SPLINE
SPL {X  -144.515, Y  +305.495, Z    +0.000, E1   +74.543, E3 +104969.530}
SPL {X  -143.690, Y  +303.925, Z    +0.000, E1   +73.372, E3 +104980.269}
SPL {X  -141.993, Y  +300.823, Z    +0.000, E1   +72.659, E3 +104987.693}
SPL {X  -138.166, Y  +294.358, Z    +0.000, E1   +72.281, E3 +104994.155}
SPL {X  -134.385, Y  +288.571, Z    +0.000, E1   +71.826, E3 +105000.418}
SPL {X  -129.872, Y  +282.297, Z    +0.000, E1   +71.229, E3 +105007.588}
SPL {X  -124.448, Y  +275.510, Z    +0.000, E1   +70.509, E3 +105014.961}
SPL {X  -117.513, Y  +267.801, Z    +0.000, E1   +72.197, E3 +105012.544}
SPL {X   -63.140, Y  +230.421, Z    +0.000, E1   +55.875, E3 +105181.983}
ENDSPLINE

SPLINE
SPL {X  -130.329, Y  +282.905, Z    +0.000, E1   +55.659, E3 +105340.318}
SPL {X  -150.766, Y  +319.018, Z    +0.000, E1   +45.408, E3 +105348.811}
SPL {X  -157.479, Y  +339.138, Z    +0.000, E1   +35.556, E3 +105350.247}
SPL {X  -160.994, Y  +356.185, Z    +0.000, E1   +24.373, E3 +105352.293}
SPL {X  -162.352, Y  +368.168, Z    +0.000, E1   +14.282, E3 +105352.345}
SPL {X  -162.808, Y  +378.562, Z    +0.000, E1    +4.298, E3 +105352.277}
SPL {X  -162.820, Y  +382.500, Z    +0.000, E1    +0.000, E3 +105351.850}
SPL {X  -162.820, Y  +384.915, Z    +0.000, E1    -4.894, E3 +105351.563}
SPL {X  -162.820, Y  +388.986, Z    +0.000, E1   -15.047, E3 +105351.661}
SPL {X  -162.820, Y  +394.732, Z    +0.000, E1   -28.992, E3 +105351.512}
SPL {X  -162.820, Y  +403.075, Z    +0.000, E1   -46.096, E3 +105351.742}
SPL {X  -162.820, Y  +414.705, Z    +0.000, E1   -61.052, E3 +105351.188}
SPL {X  -162.820, Y  +466.149, Z    +0.000, E1   -74.732, E3 +105361.185}
SPL {X  -160.722, Y  +699.554, Z    +0.000, E1   -75.485, E3 +105458.595}
SPL {X  -159.966, Y  +703.854, Z    +0.000, E1   -74.386, E3 +105473.498}
SPL {X  -156.868, Y  +717.123, Z    +0.000, E1   -74.182, E3 +105483.176}
SPL {X  -153.226, Y  +728.564, Z    +0.000, E1   -73.755, E3 +105494.184}
SPL {X  -149.090, Y  +738.941, Z    +0.000, E1   -73.348, E3 +105503.758}
SPL {X  -145.714, Y  +746.149, Z    +0.000, E1   -72.951, E3 +105511.345}
SPL {X  -140.946, Y  +755.015, Z    +0.000, E1   -72.452, E3 +105520.447}
SPL {X  -136.902, Y  +761.638, Z    +0.000, E1   -71.857, E3 +105528.314}
SPL {X  -133.350, Y  +766.925, Z    +0.000, E1   -71.498, E3 +105533.635}
SPL {X  -129.687, Y  +771.946, Z    +0.000, E1   -71.061, E3 +105539.001}
SPL {X  -126.374, Y  +776.164, Z    +0.000, E1   -70.494, E3 +105544.254}
SPL {X  -122.717, Y  +780.508, Z    +0.000, E1   -70.361, E3 +105547.292}
SPL {X  -114.093, Y  +789.660, Z    +0.000, E1   -71.634, E3 +105547.310}
SPL {X   -61.593, Y  +824.220, Z    +0.000, E1   -55.970, E3 +105713.146}
ENDSPLINE

SPLINE
SPL {X  -131.598, Y  +769.376, Z    +0.000, E1   -56.871, E3 +105879.418}
SPL {X  -152.760, Y  +729.846, Z    +0.000, E1   -44.713, E3 +105886.470}
SPL {X  -158.868, Y  +709.157, Z    +0.000, E1   -33.466, E3 +105887.671}
SPL {X  -161.987, Y  +689.949, Z    +0.000, E1   -18.777, E3 +105888.632}
SPL {X  -162.803, Y  +675.860, Z    +0.000, E1    -4.958, E3 +105888.614}
SPL {X  -162.820, Y  +671.500, Z    +0.000, E1    +0.000, E3 +105888.151}
SPL {X  -162.820, Y  +669.410, Z    +0.000, E1    +4.515, E3 +105887.913}
SPL {X  -162.820, Y  +664.781, Z    +0.000, E1   +16.411, E3 +105887.908}
SPL {X  -162.820, Y  +659.650, Z    +0.000, E1   +29.778, E3 +105887.918}
SPL {X  -162.820, Y  +651.175, Z    +0.000, E1   +47.162, E3 +105888.068}
SPL {X  -162.820, Y  +637.134, Z    +0.000, E1   +65.232, E3 +105886.610}
SPL {X  -162.820, Y  +616.721, Z    +0.000, E1   +72.273, E3 +105890.344}
SPL {X  -162.820, Y  +577.172, Z    +0.000, E1   +75.843, E3 +105900.324}
SPL {X  -159.895, Y  +349.775, Z    +0.000, E1   +76.042, E3 +105991.990}
ENDSPLINE

SPLINE
SPL {X  -160.357, Y  +352.285, Z    +0.000, E1   +74.783, E3 +106004.928}
ENDSPLINE

SPLINE
SPL {X  -145.737, Y  +307.897, Z    +0.000, E1   +77.368, E3 +105997.503}
SPL {X  -145.329, Y  +307.084, Z    +0.000, E1   +76.571, E3 +106006.340}
ENDSPLINE

SPLINE
SPL {X  -145.355, Y  +307.136, Z    +0.000, E1   +75.607, E3 +106015.864}
ENDSPLINE

SPLINE
SPL {X  -144.515, Y  +305.495, Z    +0.000, E1   +74.543, E3 +106026.673}
SPL {X  -143.702, Y  +303.949, Z    +0.000, E1   +73.349, E3 +106037.595}
ENDSPLINE

SPLINE
SPL {X  -148.050, Y  +312.738, Z    +0.000, E1   +70.533, E3 +106054.970}
ENDSPLINE

SPLINE
SPL {X  -143.809, Y  +304.150, Z    +0.000, E1   +70.034, E3 +106064.386}
SPL {X  -139.938, Y  +297.268, Z    +0.000, E1   +69.438, E3 +106072.977}
SPL {X  -136.192, Y  +291.270, Z    +0.000, E1   +68.926, E3 +106080.124}
SPL {X  -131.963, Y  +285.127, Z    +0.000, E1   +68.405, E3 +106087.114}
SPL {X  -127.466, Y  +279.195, Z    +0.000, E1   +67.714, E3 +106094.402}
SPL {X  -119.204, Y  +269.591, Z    +0.000, E1   +69.726, E3 +106092.393}
SPL {X   -73.382, Y  +235.154, Z    +0.000, E1   +54.977, E3 +106258.070}
ENDSPLINE

SPLINE
SPL {X  -133.875, Y  +287.830, Z    +0.000, E1   +51.751, E3 +106397.273}
SPL {X  -153.240, Y  +325.474, Z    +0.000, E1   +39.999, E3 +106408.476}
SPL {X  -159.032, Y  +345.583, Z    +0.000, E1   +29.156, E3 +106408.960}
SPL {X  -161.304, Y  +358.334, Z    +0.000, E1   +20.524, E3 +106408.917}
SPL {X  -162.437, Y  +369.334, Z    +0.000, E1   +11.998, E3 +106410.096}
SPL {X  -162.814, Y  +379.161, Z    +0.000, E1    +3.343, E3 +106410.115}
SPL {X  -162.820, Y  +382.500, Z    +0.000, E1    +0.000, E3 +106409.598}
SPL {X  -162.820, Y  +384.390, Z    +0.000, E1    -3.279, E3 +106409.315}
SPL {X  -162.820, Y  +388.496, Z    +0.000, E1   -11.991, E3 +106409.217}
SPL {X  -162.820, Y  +392.944, Z    +0.000, E1   -22.020, E3 +106409.242}
SPL {X  -162.820, Y  +397.954, Z    +0.000, E1   -32.843, E3 +106409.282}
SPL {X  -162.820, Y  +404.232, Z    +0.000, E1   -44.157, E3 +106409.290}
SPL {X  -162.820, Y  +415.904, Z    +0.000, E1   -58.030, E3 +106409.563}
SPL {X  -162.820, Y  +472.155, Z    +0.000, E1   -74.123, E3 +106419.666}
SPL {X  -162.820, Y  +661.743, Z    +0.000, E1   -73.395, E3 +106514.800}
ENDSPLINE

SPLINE
SPL {X  -162.820, Y  +658.105, Z    +0.000, E1   -71.889, E3 +106528.198}
ENDSPLINE

SPLINE
SPL {X  -162.784, Y  +676.927, Z    +0.000, E1   -71.815, E3 +106541.726}
SPL {X  -161.514, Y  +694.081, Z    +0.000, E1   -71.845, E3 +106553.116}
SPL {X  -159.782, Y  +704.807, Z    +0.000, E1   -71.464, E3 +106564.098}
SPL {X  -157.050, Y  +716.463, Z    +0.000, E1   -71.316, E3 +106573.398}
SPL {X  -154.424, Y  +725.109, Z    +0.000, E1   -70.982, E3 +106582.250}
SPL {X  -151.195, Y  +733.918, Z    +0.000, E1   -70.611, E3 +106591.372}
SPL {X  -147.776, Y  +741.856, Z    +0.000, E1   -70.224, E3 +106599.820}
SPL {X  -144.623, Y  +748.297, Z    +0.000, E1   -69.772, E3 +106607.445}
SPL {X  -141.153, Y  +754.655, Z    +0.000, E1   -69.344, E3 +106614.749}
SPL {X  -137.365, Y  +760.914, Z    +0.000, E1   -68.751, E3 +106622.687}
SPL {X  -133.334, Y  +766.947, Z    +0.000, E1   -68.226, E3 +106629.792}
SPL {X  -129.138, Y  +772.665, Z    +0.000, E1   -67.631, E3 +106636.599}
SPL {X  -125.533, Y  +777.190, Z    +0.000, E1   -67.475, E3 +106640.296}
SPL {X   -73.826, Y  +818.621, Z    +0.000, E1   -58.574, E3 +106735.789}
ENDSPLINE

SPLINE
SPL {X  -110.901, Y  +792.711, Z    +0.000, E1   -55.300, E3 +106920.647}
SPL {X  -144.508, Y  +748.519, Z    +0.000, E1   -46.961, E3 +106945.683}
SPL {X  -158.446, Y  +710.986, Z    +0.000, E1   -30.228, E3 +106949.049}
SPL {X  -162.035, Y  +689.470, Z    +0.000, E1   -15.657, E3 +106950.620}
SPL {X  -162.788, Y  +676.746, Z    +0.000, E1    -5.020, E3 +106950.527}
SPL {X  -162.820, Y  +671.525, Z    +0.000, E1    -0.042, E3 +106950.081}
SPL {X  -162.820, Y  +669.531, Z    +0.000, E1    +3.299, E3 +106949.770}
SPL {X  -162.820, Y  +664.807, Z    +0.000, E1   +13.064, E3 +106949.699}
SPL {X  -162.820, Y  +659.610, Z    +0.000, E1   +24.615, E3 +106949.680}
SPL {X  -162.820, Y  +651.281, Z    +0.000, E1   +40.220, E3 +106950.233}
SPL {X  -162.820, Y  +632.362, Z    +0.000, E1   +62.930, E3 +106948.892}
SPL {X  -162.820, Y  +579.681, Z    +0.000, E1   +72.301, E3 +106964.678}
SPL {X  -162.820, Y  +402.073, Z    +0.000, E1   +73.274, E3 +107050.213}
ENDSPLINE

SPLINE
SPL {X  -162.820, Y  +412.258, Z    +0.000, E1   +71.454, E3 +107061.310}
SPL {X  -162.820, Y  +452.249, Z    +0.000, E1   +66.666, E3 +107073.116}
ENDSPLINE

SPLINE
SPL {X  -162.820, Y  +427.408, Z    +0.000, E1   +67.534, E3 +107087.734}
SPL {X  -162.820, Y  +409.075, Z    +0.000, E1   +68.145, E3 +107098.119}
SPL {X  -162.820, Y  +384.968, Z    +0.000, E1   +68.973, E3 +107110.678}
SPL {X  -162.073, Y  +364.922, Z    +0.000, E1   +69.599, E3 +107120.804}
SPL {X  -158.958, Y  +345.247, Z    +0.000, E1   +70.087, E3 +107131.400}
SPL {X  -152.677, Y  +323.931, Z    +0.000, E1   +70.710, E3 +107141.161}
SPL {X  -148.063, Y  +312.768, Z    +0.000, E1   +70.492, E3 +107150.482}
SPL {X  -143.809, Y  +304.150, Z    +0.000, E1   +70.034, E3 +107159.625}
SPL {X  -139.938, Y  +297.268, Z    +0.000, E1   +69.438, E3 +107168.215}
SPL {X  -136.192, Y  +291.270, Z    +0.000, E1   +68.926, E3 +107175.362}
SPL {X  -131.963, Y  +285.127, Z    +0.000, E1   +68.405, E3 +107182.352}
SPL {X  -127.466, Y  +279.195, Z    +0.000, E1   +67.714, E3 +107189.640}
SPL {X  -119.204, Y  +269.591, Z    +0.000, E1   +69.726, E3 +107187.631}
SPL {X   -73.382, Y  +235.154, Z    +0.000, E1   +54.977, E3 +107353.308}
ENDSPLINE

SPLINE
SPL {X  -133.875, Y  +287.830, Z    +0.000, E1   +51.751, E3 +107492.511}
SPL {X  -153.240, Y  +325.474, Z    +0.000, E1   +39.999, E3 +107503.714}
SPL {X  -160.567, Y  +353.506, Z    +0.000, E1   +24.043, E3 +107504.208}
SPL {X  -162.437, Y  +369.334, Z    +0.000, E1   +11.998, E3 +107505.334}
SPL {X  -162.814, Y  +379.161, Z    +0.000, E1    +3.343, E3 +107505.353}
SPL {X  -162.820, Y  +382.751, Z    +0.000, E1    -0.252, E3 +107504.767}
SPL {X  -162.820, Y  +387.406, Z    +0.000, E1    -9.377, E3 +107504.488}
SPL {X  -162.820, Y  +392.944, Z    +0.000, E1   -22.020, E3 +107504.480}
SPL {X  -162.820, Y  +397.954, Z    +0.000, E1   -32.843, E3 +107504.520}
SPL {X  -162.820, Y  +404.232, Z    +0.000, E1   -44.157, E3 +107504.528}
SPL {X  -162.820, Y  +415.904, Z    +0.000, E1   -58.030, E3 +107504.801}
SPL {X  -162.820, Y  +472.155, Z    +0.000, E1   -74.123, E3 +107514.904}
SPL {X  -162.820, Y  +661.743, Z    +0.000, E1   -73.395, E3 +107610.038}
ENDSPLINE

SPLINE
SPL {X  -162.820, Y  +658.105, Z    +0.000, E1   -71.889, E3 +107623.436}
ENDSPLINE

SPLINE
SPL {X  -162.784, Y  +676.927, Z    +0.000, E1   -71.815, E3 +107636.964}
SPL {X  -161.514, Y  +694.081, Z    +0.000, E1   -71.845, E3 +107648.354}
SPL {X  -159.782, Y  +704.807, Z    +0.000, E1   -71.464, E3 +107659.336}
SPL {X  -157.050, Y  +716.463, Z    +0.000, E1   -71.316, E3 +107668.636}
SPL {X  -154.424, Y  +725.109, Z    +0.000, E1   -70.982, E3 +107677.488}
SPL {X  -151.195, Y  +733.918, Z    +0.000, E1   -70.611, E3 +107686.610}
SPL {X  -147.776, Y  +741.856, Z    +0.000, E1   -70.224, E3 +107695.059}
SPL {X  -143.411, Y  +750.594, Z    +0.000, E1   -69.653, E3 +107705.215}
SPL {X  -138.205, Y  +759.580, Z    +0.000, E1   -68.913, E3 +107716.164}
SPL {X  -133.334, Y  +766.947, Z    +0.000, E1   -68.226, E3 +107725.030}
SPL {X  -129.138, Y  +772.665, Z    +0.000, E1   -67.631, E3 +107731.837}
SPL {X  -125.533, Y  +777.190, Z    +0.000, E1   -67.475, E3 +107735.534}
SPL {X   -73.826, Y  +818.621, Z    +0.000, E1   -58.574, E3 +107831.027}
ENDSPLINE

SPLINE
SPL {X  -110.901, Y  +792.711, Z    +0.000, E1   -55.300, E3 +108015.885}
SPL {X  -144.508, Y  +748.519, Z    +0.000, E1   -46.961, E3 +108040.922}
SPL {X  -156.638, Y  +717.940, Z    +0.000, E1   -34.002, E3 +108043.657}
SPL {X  -160.830, Y  +698.875, Z    +0.000, E1   -22.517, E3 +108045.321}
SPL {X  -162.277, Y  +686.786, Z    +0.000, E1   -13.481, E3 +108045.900}
SPL {X  -162.788, Y  +676.746, Z    +0.000, E1    -5.020, E3 +108045.765}
SPL {X  -162.820, Y  +671.525, Z    +0.000, E1    -0.042, E3 +108045.319}
SPL {X  -162.820, Y  +670.529, Z    +0.000, E1    +1.628, E3 +108045.021}
SPL {X  -162.820, Y  +667.499, Z    +0.000, E1    +7.374, E3 +108045.010}
SPL {X  -162.820, Y  +663.777, Z    +0.000, E1   +15.496, E3 +108044.873}
SPL {X  -162.820, Y  +659.610, Z    +0.000, E1   +24.615, E3 +108044.918}
SPL {X  -162.820, Y  +651.281, Z    +0.000, E1   +40.220, E3 +108045.471}
SPL {X  -162.820, Y  +632.362, Z    +0.000, E1   +62.930, E3 +108044.130}
SPL {X  -162.820, Y  +579.681, Z    +0.000, E1   +72.301, E3 +108059.917}
SPL {X  -162.820, Y  +408.049, Z    +0.000, E1   +72.202, E3 +108152.348}
ENDSPLINE

SPLINE
SPL {X  -162.820, Y  +452.249, Z    +0.000, E1   +66.666, E3 +108168.354}
ENDSPLINE

SPLINE
SPL {X  -162.820, Y  +427.408, Z    +0.000, E1   +67.534, E3 +108182.973}
SPL {X  -162.820, Y  +409.075, Z    +0.000, E1   +68.145, E3 +108193.357}
SPL {X  -162.820, Y  +384.968, Z    +0.000, E1   +68.973, E3 +108205.917}
SPL {X  -161.511, Y  +359.895, Z    +0.000, E1   +69.744, E3 +108218.653}
SPL {X  -158.246, Y  +342.178, Z    +0.000, E1   +70.136, E3 +108228.402}
SPL {X  -152.677, Y  +323.931, Z    +0.000, E1   +70.710, E3 +108236.399}
SPL {X  -148.063, Y  +312.768, Z    +0.000, E1   +70.492, E3 +108245.720}
SPL {X  -143.809, Y  +304.150, Z    +0.000, E1   +70.034, E3 +108254.863}
SPL {X  -139.938, Y  +297.268, Z    +0.000, E1   +69.438, E3 +108263.453}
SPL {X  -136.192, Y  +291.270, Z    +0.000, E1   +68.926, E3 +108270.600}
SPL {X  -131.963, Y  +285.127, Z    +0.000, E1   +68.405, E3 +108277.591}
SPL {X  -127.466, Y  +279.195, Z    +0.000, E1   +67.714, E3 +108284.878}
SPL {X  -119.204, Y  +269.591, Z    +0.000, E1   +69.726, E3 +108282.869}
SPL {X   -73.382, Y  +235.154, Z    +0.000, E1   +54.977, E3 +108448.546}
ENDSPLINE

SPLINE
SPL {X  -133.875, Y  +287.830, Z    +0.000, E1   +51.751, E3 +108587.749}
SPL {X  -153.240, Y  +325.474, Z    +0.000, E1   +39.999, E3 +108598.952}
SPL {X  -160.567, Y  +353.506, Z    +0.000, E1   +24.043, E3 +108599.446}
SPL {X  -162.646, Y  +372.968, Z    +0.000, E1    +8.995, E3 +108600.623}
SPL {X  -162.820, Y  +382.382, Z    +0.000, E1    +0.204, E3 +108600.110}
SPL {X  -162.820, Y  +384.390, Z    +0.000, E1    -3.279, E3 +108599.791}
SPL {X  -162.820, Y  +388.496, Z    +0.000, E1   -11.991, E3 +108599.693}
SPL {X  -162.820, Y  +392.944, Z    +0.000, E1   -22.020, E3 +108599.718}
SPL {X  -162.820, Y  +397.954, Z    +0.000, E1   -32.843, E3 +108599.758}
SPL {X  -162.820, Y  +404.232, Z    +0.000, E1   -44.157, E3 +108599.766}
SPL {X  -162.820, Y  +415.904, Z    +0.000, E1   -58.030, E3 +108600.039}
SPL {X  -162.820, Y  +467.484, Z    +0.000, E1   -73.355, E3 +108609.869}
SPL {X  -162.820, Y  +491.822, Z    +0.000, E1   -76.748, E3 +108611.292}
SPL {X  -162.820, Y  +661.743, Z    +0.000, E1   -73.395, E3 +108705.276}
ENDSPLINE

SPLINE
SPL {X  -162.820, Y  +658.105, Z    +0.000, E1   -71.889, E3 +108718.675}
ENDSPLINE

SPLINE
SPL {X  -162.784, Y  +676.927, Z    +0.000, E1   -71.815, E3 +108732.202}
SPL {X  -161.514, Y  +694.081, Z    +0.000, E1   -71.845, E3 +108743.592}
SPL {X  -159.782, Y  +704.807, Z    +0.000, E1   -71.464, E3 +108754.574}
SPL {X  -157.050, Y  +716.463, Z    +0.000, E1   -71.316, E3 +108763.874}
SPL {X  -154.424, Y  +725.109, Z    +0.000, E1   -70.982, E3 +108772.726}
SPL {X  -150.493, Y  +735.646, Z    +0.000, E1   -70.534, E3 +108783.771}
SPL {X  -145.565, Y  +746.446, Z    +0.000, E1   -69.958, E3 +108795.480}
SPL {X  -142.097, Y  +752.991, Z    +0.000, E1   -69.463, E3 +108803.220}
SPL {X  -138.205, Y  +759.580, Z    +0.000, E1   -68.913, E3 +108811.402}
SPL {X  -133.334, Y  +766.947, Z    +0.000, E1   -68.226, E3 +108820.268}
SPL {X  -129.943, Y  +771.607, Z    +0.000, E1   -67.755, E3 +108825.716}
SPL {X  -126.438, Y  +776.086, Z    +0.000, E1   -67.465, E3 +108830.086}
SPL {X   -73.826, Y  +818.621, Z    +0.000, E1   -58.574, E3 +108926.265}
ENDSPLINE

SPLINE
SPL {X  -110.901, Y  +792.711, Z    +0.000, E1   -55.300, E3 +109111.123}
SPL {X  -144.508, Y  +748.519, Z    +0.000, E1   -46.961, E3 +109136.160}
SPL {X  -158.446, Y  +710.986, Z    +0.000, E1   -30.228, E3 +109139.525}
SPL {X  -162.035, Y  +689.470, Z    +0.000, E1   -15.657, E3 +109141.096}
SPL {X  -162.788, Y  +676.746, Z    +0.000, E1    -5.020, E3 +109141.003}
SPL {X  -162.820, Y  +671.525, Z    +0.000, E1    -0.042, E3 +109140.557}
SPL {X  -162.820, Y  +669.531, Z    +0.000, E1    +3.299, E3 +109140.246}
SPL {X  -162.820, Y  +664.807, Z    +0.000, E1   +13.064, E3 +109140.175}
SPL {X  -162.820, Y  +659.610, Z    +0.000, E1   +24.615, E3 +109140.156}
SPL {X  -162.820, Y  +654.471, Z    +0.000, E1   +35.284, E3 +109140.058}
SPL {X  -162.820, Y  +648.111, Z    +0.000, E1   +44.823, E3 +109141.355}
SPL {X  -162.820, Y  +635.984, Z    +0.000, E1   +61.208, E3 +109138.363}
SPL {X  -162.820, Y  +617.261, Z    +0.000, E1   +67.803, E3 +109143.550}
SPL {X  -162.820, Y  +579.681, Z    +0.000, E1   +72.301, E3 +109155.155}
SPL {X  -162.820, Y  +408.049, Z    +0.000, E1   +72.202, E3 +109247.586}
ENDSPLINE

SPLINE
SPL {X  -162.820, Y  +452.249, Z    +0.000, E1   +66.666, E3 +109263.592}
ENDSPLINE

SPLINE
SPL {X  -162.820, Y  +427.408, Z    +0.000, E1   +67.534, E3 +109278.211}
SPL {X  -162.820, Y  +402.068, Z    +0.000, E1   +68.403, E3 +109292.272}
SPL {X  -162.523, Y  +370.677, Z    +0.000, E1   +69.437, E3 +109308.333}
SPL {X  -158.958, Y  +345.247, Z    +0.000, E1   +70.087, E3 +109321.876}
SPL {X  -154.257, Y  +328.393, Z    +0.000, E1   +70.602, E3 +109329.433}
SPL {X  -150.447, Y  +318.243, Z    +0.000, E1   +70.683, E3 +109335.779}
SPL {X  -145.895, Y  +308.216, Z    +0.000, E1   +70.273, E3 +109345.732}
SPL {X  -140.654, Y  +298.483, Z    +0.000, E1   +69.615, E3 +109356.874}
SPL {X  -136.192, Y  +291.270, Z    +0.000, E1   +68.926, E3 +109365.838}
SPL {X  -131.963, Y  +285.127, Z    +0.000, E1   +68.405, E3 +109372.829}
SPL {X  -127.466, Y  +279.195, Z    +0.000, E1   +67.714, E3 +109380.116}
SPL {X  -119.204, Y  +269.591, Z    +0.000, E1   +69.726, E3 +109378.108}
SPL {X   -73.382, Y  +235.154, Z    +0.000, E1   +54.977, E3 +109543.785}
ENDSPLINE

SPLINE
SPL {X  -115.538, Y  +265.778, Z    +0.000, E1   +55.826, E3 +109674.236}
SPL {X  -140.740, Y  +298.630, Z    +0.000, E1   +48.901, E3 +109685.571}
SPL {X  -153.240, Y  +325.474, Z    +0.000, E1   +39.999, E3 +109694.190}
SPL {X  -159.032, Y  +345.583, Z    +0.000, E1   +29.156, E3 +109694.674}
SPL {X  -161.304, Y  +358.334, Z    +0.000, E1   +20.524, E3 +109694.631}
SPL {X  -162.646, Y  +372.968, Z    +0.000, E1    +8.995, E3 +109695.861}
SPL {X  -162.820, Y  +382.646, Z    +0.000, E1    -0.044, E3 +109695.275}
SPL {X  -162.820, Y  +387.406, Z    +0.000, E1    -9.377, E3 +109694.965}
SPL {X  -162.820, Y  +392.944, Z    +0.000, E1   -22.020, E3 +109694.956}
SPL {X  -162.820, Y  +397.954, Z    +0.000, E1   -32.843, E3 +109694.996}
SPL {X  -162.820, Y  +404.232, Z    +0.000, E1   -44.157, E3 +109695.004}
SPL {X  -162.820, Y  +415.904, Z    +0.000, E1   -58.030, E3 +109695.278}
SPL {X  -162.820, Y  +472.155, Z    +0.000, E1   -74.123, E3 +109705.380}
SPL {X  -162.820, Y  +654.572, Z    +0.000, E1   -72.288, E3 +109807.606}
SPL {X  -162.820, Y  +673.151, Z    +0.000, E1   -71.906, E3 +109824.175}
SPL {X  -161.514, Y  +694.081, Z    +0.000, E1   -71.845, E3 +109838.830}
SPL {X  -159.782, Y  +704.807, Z    +0.000, E1   -71.464, E3 +109849.812}
SPL {X  -157.050, Y  +716.463, Z    +0.000, E1   -71.316, E3 +109859.112}
SPL {X  -154.424, Y  +725.109, Z    +0.000, E1   -70.982, E3 +109867.964}
SPL {X  -150.493, Y  +735.646, Z    +0.000, E1   -70.534, E3 +109879.009}
SPL {X  -145.565, Y  +746.446, Z    +0.000, E1   -69.958, E3 +109890.718}
SPL {X  -141.153, Y  +754.655, Z    +0.000, E1   -69.344, E3 +109900.463}
SPL {X  -137.365, Y  +760.914, Z    +0.000, E1   -68.751, E3 +109908.401}
SPL {X  -133.334, Y  +766.947, Z    +0.000, E1   -68.226, E3 +109915.506}
SPL {X  -129.943, Y  +771.607, Z    +0.000, E1   -67.755, E3 +109920.954}
SPL {X  -126.438, Y  +776.086, Z    +0.000, E1   -67.465, E3 +109925.324}
SPL {X   -73.826, Y  +818.621, Z    +0.000, E1   -58.574, E3 +110021.503}
ENDSPLINE

SPLINE
SPL {X  -110.901, Y  +792.711, Z    +0.000, E1   -55.300, E3 +110206.361}
SPL {X  -144.508, Y  +748.519, Z    +0.000, E1   -46.961, E3 +110231.398}
SPL {X  -158.446, Y  +710.986, Z    +0.000, E1   -30.228, E3 +110234.763}
SPL {X  -162.035, Y  +689.470, Z    +0.000, E1   -15.657, E3 +110236.334}
SPL {X  -162.696, Y  +679.865, Z    +0.000, E1    -7.693, E3 +110236.406}
SPL {X  -162.820, Y  +671.472, Z    +0.000, E1    -0.171, E3 +110235.745}
SPL {X  -162.820, Y  +667.499, Z    +0.000, E1    +7.374, E3 +110235.486}
SPL {X  -162.820, Y  +663.777, Z    +0.000, E1   +15.496, E3 +110235.349}
SPL {X  -162.820, Y  +659.610, Z    +0.000, E1   +24.615, E3 +110235.394}
SPL {X  -162.820, Y  +654.471, Z    +0.000, E1   +35.284, E3 +110235.296}
SPL {X  -162.820, Y  +648.111, Z    +0.000, E1   +44.823, E3 +110236.593}
SPL {X  -162.820, Y  +635.984, Z    +0.000, E1   +61.208, E3 +110233.601}
SPL {X  -162.820, Y  +617.261, Z    +0.000, E1   +67.803, E3 +110238.788}
SPL {X  -162.820, Y  +579.681, Z    +0.000, E1   +72.301, E3 +110250.393}
SPL {X  -162.820, Y  +408.049, Z    +0.000, E1   +72.202, E3 +110342.825}
ENDSPLINE

SPLINE
SPL {X  -162.820, Y  +452.249, Z    +0.000, E1   +66.666, E3 +110358.830}
ENDSPLINE

SPLINE
SPL {X  -162.820, Y  +427.408, Z    +0.000, E1   +67.534, E3 +110373.449}
SPL {X  -162.820, Y  +402.068, Z    +0.000, E1   +68.403, E3 +110387.510}
SPL {X  -162.804, Y  +378.229, Z    +0.000, E1   +69.183, E3 +110399.837}
SPL {X  -161.511, Y  +359.895, Z    +0.000, E1   +69.744, E3 +110409.129}
SPL {X  -158.246, Y  +342.178, Z    +0.000, E1   +70.136, E3 +110418.878}
SPL {X  -152.677, Y  +323.931, Z    +0.000, E1   +70.710, E3 +110426.875}
SPL {X  -148.063, Y  +312.768, Z    +0.000, E1   +70.492, E3 +110436.196}
SPL {X  -143.809, Y  +304.150, Z    +0.000, E1   +70.034, E3 +110445.339}
SPL {X  -139.938, Y  +297.268, Z    +0.000, E1   +69.438, E3 +110453.929}
SPL {X  -136.192, Y  +291.270, Z    +0.000, E1   +68.926, E3 +110461.076}
SPL {X  -131.963, Y  +285.127, Z    +0.000, E1   +68.405, E3 +110468.067}
SPL {X  -127.466, Y  +279.195, Z    +0.000, E1   +67.714, E3 +110475.354}
SPL {X  -119.204, Y  +269.591, Z    +0.000, E1   +69.726, E3 +110473.346}
SPL {X   -73.382, Y  +235.154, Z    +0.000, E1   +54.977, E3 +110639.023}
ENDSPLINE

SPLINE
SPL {X  -115.538, Y  +265.778, Z    +0.000, E1   +55.826, E3 +110769.474}
SPL {X  -140.740, Y  +298.630, Z    +0.000, E1   +48.901, E3 +110780.809}
SPL {X  -153.240, Y  +325.474, Z    +0.000, E1   +39.999, E3 +110789.428}
SPL {X  -159.032, Y  +345.583, Z    +0.000, E1   +29.156, E3 +110789.912}
SPL {X  -161.304, Y  +358.334, Z    +0.000, E1   +20.524, E3 +110789.870}
SPL {X  -162.437, Y  +369.334, Z    +0.000, E1   +11.998, E3 +110791.048}
SPL {X  -162.814, Y  +379.161, Z    +0.000, E1    +3.343, E3 +110791.068}
SPL {X  -162.820, Y  +382.751, Z    +0.000, E1    -0.252, E3 +110790.482}
SPL {X  -162.820, Y  +387.406, Z    +0.000, E1    -9.377, E3 +110790.203}
SPL {X  -162.820, Y  +392.944, Z    +0.000, E1   -22.020, E3 +110790.194}
SPL {X  -162.820, Y  +397.954, Z    +0.000, E1   -32.843, E3 +110790.234}
SPL {X  -162.820, Y  +404.232, Z    +0.000, E1   -44.157, E3 +110790.242}
SPL {X  -162.820, Y  +415.904, Z    +0.000, E1   -58.030, E3 +110790.516}
SPL {X  -162.820, Y  +467.484, Z    +0.000, E1   -73.355, E3 +110800.345}
SPL {X  -162.820, Y  +491.822, Z    +0.000, E1   -76.748, E3 +110801.768}
SPL {X  -162.820, Y  +661.743, Z    +0.000, E1   -73.395, E3 +110895.753}
ENDSPLINE

SPLINE
SPL {X  -162.820, Y  +658.105, Z    +0.000, E1   -71.889, E3 +110909.151}
ENDSPLINE

SPLINE
SPL {X  -162.784, Y  +676.927, Z    +0.000, E1   -71.815, E3 +110922.679}
SPL {X  -161.514, Y  +694.081, Z    +0.000, E1   -71.845, E3 +110934.068}
SPL {X  -159.782, Y  +704.807, Z    +0.000, E1   -71.464, E3 +110945.051}
SPL {X  -157.050, Y  +716.463, Z    +0.000, E1   -71.316, E3 +110954.350}
SPL {X  -154.424, Y  +725.109, Z    +0.000, E1   -70.982, E3 +110963.202}
SPL {X  -150.493, Y  +735.646, Z    +0.000, E1   -70.534, E3 +110974.247}
SPL {X  -145.565, Y  +746.446, Z    +0.000, E1   -69.958, E3 +110985.956}
SPL {X  -141.153, Y  +754.655, Z    +0.000, E1   -69.344, E3 +110995.701}
SPL {X  -137.365, Y  +760.914, Z    +0.000, E1   -68.751, E3 +111003.639}
SPL {X  -133.334, Y  +766.947, Z    +0.000, E1   -68.226, E3 +111010.744}
SPL {X  -129.138, Y  +772.665, Z    +0.000, E1   -67.631, E3 +111017.551}
SPL {X  -125.533, Y  +777.190, Z    +0.000, E1   -67.475, E3 +111021.249}
SPL {X   -73.826, Y  +818.621, Z    +0.000, E1   -58.574, E3 +111116.742}
ENDSPLINE

SPLINE
SPL {X  -110.901, Y  +792.711, Z    +0.000, E1   -55.300, E3 +111301.599}
SPL {X  -144.508, Y  +748.519, Z    +0.000, E1   -46.961, E3 +111326.636}
SPL {X  -156.638, Y  +717.940, Z    +0.000, E1   -34.002, E3 +111329.372}
SPL {X  -160.830, Y  +698.875, Z    +0.000, E1   -22.517, E3 +111331.035}
SPL {X  -162.277, Y  +686.786, Z    +0.000, E1   -13.481, E3 +111331.614}
SPL {X  -162.788, Y  +676.746, Z    +0.000, E1    -5.020, E3 +111331.479}
SPL {X  -162.820, Y  +671.525, Z    +0.000, E1    -0.042, E3 +111331.034}
SPL {X  -162.820, Y  +669.531, Z    +0.000, E1    +3.299, E3 +111330.722}
SPL {X  -162.820, Y  +664.807, Z    +0.000, E1   +13.064, E3 +111330.651}
SPL {X  -162.820, Y  +659.610, Z    +0.000, E1   +24.615, E3 +111330.632}
SPL {X  -162.820, Y  +654.471, Z    +0.000, E1   +35.284, E3 +111330.534}
SPL {X  -162.820, Y  +648.111, Z    +0.000, E1   +44.823, E3 +111331.831}
SPL {X  -162.820, Y  +635.984, Z    +0.000, E1   +61.208, E3 +111328.839}
SPL {X  -162.820, Y  +617.261, Z    +0.000, E1   +67.803, E3 +111334.026}
SPL {X  -162.820, Y  +579.681, Z    +0.000, E1   +72.301, E3 +111345.631}
SPL {X  -162.820, Y  +408.049, Z    +0.000, E1   +72.202, E3 +111438.063}
ENDSPLINE

SPLINE
SPL {X  -162.820, Y  +452.249, Z    +0.000, E1   +66.666, E3 +111454.068}
ENDSPLINE

SPLINE
SPL {X  -162.820, Y  +427.408, Z    +0.000, E1   +67.534, E3 +111468.687}
SPL {X  -162.820, Y  +402.068, Z    +0.000, E1   +68.403, E3 +111482.748}
SPL {X  -162.523, Y  +370.677, Z    +0.000, E1   +69.437, E3 +111498.809}
SPL {X  -158.958, Y  +345.247, Z    +0.000, E1   +70.087, E3 +111512.352}
SPL {X  -154.257, Y  +328.393, Z    +0.000, E1   +70.602, E3 +111519.909}
SPL {X  -150.447, Y  +318.243, Z    +0.000, E1   +70.683, E3 +111526.255}
SPL {X  -145.895, Y  +308.216, Z    +0.000, E1   +70.273, E3 +111536.208}
SPL {X  -140.654, Y  +298.483, Z    +0.000, E1   +69.615, E3 +111547.350}
SPL {X  -136.192, Y  +291.270, Z    +0.000, E1   +68.926, E3 +111556.314}
SPL {X  -131.963, Y  +285.127, Z    +0.000, E1   +68.405, E3 +111563.305}
SPL {X  -127.466, Y  +279.195, Z    +0.000, E1   +67.714, E3 +111570.592}
SPL {X  -119.204, Y  +269.591, Z    +0.000, E1   +69.726, E3 +111568.584}
SPL {X   -73.382, Y  +235.154, Z    +0.000, E1   +54.977, E3 +111734.261}
ENDSPLINE

SPLINE
SPL {X  -115.538, Y  +265.778, Z    +0.000, E1   +55.826, E3 +111864.712}
SPL {X  -140.740, Y  +298.630, Z    +0.000, E1   +48.901, E3 +111876.047}
SPL {X  -153.240, Y  +325.474, Z    +0.000, E1   +39.999, E3 +111884.666}
SPL {X  -159.032, Y  +345.583, Z    +0.000, E1   +29.156, E3 +111885.150}
SPL {X  -161.304, Y  +358.334, Z    +0.000, E1   +20.524, E3 +111885.108}
SPL {X  -162.646, Y  +372.968, Z    +0.000, E1    +8.995, E3 +111886.337}
SPL {X  -162.820, Y  +382.382, Z    +0.000, E1    +0.204, E3 +111885.824}
SPL {X  -162.820, Y  +384.390, Z    +0.000, E1    -3.279, E3 +111885.505}
SPL {X  -162.820, Y  +388.496, Z    +0.000, E1   -11.991, E3 +111885.407}
SPL {X  -162.820, Y  +392.944, Z    +0.000, E1   -22.020, E3 +111885.432}
SPL {X  -162.820, Y  +397.954, Z    +0.000, E1   -32.843, E3 +111885.472}
SPL {X  -162.820, Y  +404.232, Z    +0.000, E1   -44.157, E3 +111885.480}
SPL {X  -162.820, Y  +415.904, Z    +0.000, E1   -58.030, E3 +111885.754}
SPL {X  -162.820, Y  +472.155, Z    +0.000, E1   -74.123, E3 +111895.857}
SPL {X  -162.820, Y  +661.743, Z    +0.000, E1   -73.395, E3 +111990.991}
ENDSPLINE

SPLINE
SPL {X  -162.820, Y  +658.105, Z    +0.000, E1   -71.889, E3 +112004.389}
ENDSPLINE

SPLINE
SPL {X  -162.784, Y  +676.927, Z    +0.000, E1   -71.815, E3 +112017.917}
SPL {X  -161.514, Y  +694.081, Z    +0.000, E1   -71.845, E3 +112029.306}
SPL {X  -159.782, Y  +704.807, Z    +0.000, E1   -71.464, E3 +112040.289}
SPL {X  -157.050, Y  +716.463, Z    +0.000, E1   -71.316, E3 +112049.588}
SPL {X  -154.424, Y  +725.109, Z    +0.000, E1   -70.982, E3 +112058.440}
SPL {X  -151.195, Y  +733.918, Z    +0.000, E1   -70.611, E3 +112067.563}
SPL {X  -147.776, Y  +741.856, Z    +0.000, E1   -70.224, E3 +112076.011}
SPL {X  -144.623, Y  +748.297, Z    +0.000, E1   -69.772, E3 +112083.636}
SPL {X  -141.153, Y  +754.655, Z    +0.000, E1   -69.344, E3 +112090.939}
SPL {X  -136.484, Y  +762.283, Z    +0.000, E1   -68.639, E3 +112100.572}
SPL {X  -132.373, Y  +768.304, Z    +0.000, E1   -68.109, E3 +112107.442}
SPL {X  -129.138, Y  +772.665, Z    +0.000, E1   -67.631, E3 +112112.789}
SPL {X  -125.533, Y  +777.190, Z    +0.000, E1   -67.475, E3 +112116.487}
SPL {X   -73.826, Y  +818.621, Z    +0.000, E1   -58.574, E3 +112211.980}
ENDSPLINE

SPLINE
SPL {X  -110.901, Y  +792.711, Z    +0.000, E1   -55.300, E3 +112396.837}
SPL {X  -144.508, Y  +748.519, Z    +0.000, E1   -46.961, E3 +112421.874}
SPL {X  -156.638, Y  +717.940, Z    +0.000, E1   -34.002, E3 +112424.610}
SPL {X  -160.830, Y  +698.875, Z    +0.000, E1   -22.517, E3 +112426.273}
SPL {X  -162.532, Y  +683.174, Z    +0.000, E1   -10.600, E3 +112426.879}
SPL {X  -162.815, Y  +674.755, Z    +0.000, E1    -3.125, E3 +112426.603}
SPL {X  -162.820, Y  +671.525, Z    +0.000, E1    -0.042, E3 +112426.272}
SPL {X  -162.820, Y  +670.529, Z    +0.000, E1    +1.628, E3 +112425.973}
SPL {X  -162.820, Y  +667.499, Z    +0.000, E1    +7.374, E3 +112425.962}
SPL {X  -162.820, Y  +663.777, Z    +0.000, E1   +15.496, E3 +112425.825}
SPL {X  -162.820, Y  +659.610, Z    +0.000, E1   +24.615, E3 +112425.870}
SPL {X  -162.820, Y  +651.281, Z    +0.000, E1   +40.220, E3 +112426.423}
SPL {X  -162.820, Y  +632.362, Z    +0.000, E1   +62.930, E3 +112425.083}
SPL {X  -162.820, Y  +579.681, Z    +0.000, E1   +72.301, E3 +112440.869}
SPL {X  -162.820, Y  +408.049, Z    +0.000, E1   +72.202, E3 +112533.301}
ENDSPLINE

SPLINE
SPL {X  -162.820, Y  +452.249, Z    +0.000, E1   +66.666, E3 +112549.306}
ENDSPLINE

SPLINE
SPL {X  -162.820, Y  +427.408, Z    +0.000, E1   +67.534, E3 +112563.925}
SPL {X  -162.820, Y  +402.068, Z    +0.000, E1   +68.403, E3 +112577.986}
SPL {X  -162.523, Y  +370.677, Z    +0.000, E1   +69.437, E3 +112594.047}
SPL {X  -158.958, Y  +345.247, Z    +0.000, E1   +70.087, E3 +112607.590}
SPL {X  -152.677, Y  +323.931, Z    +0.000, E1   +70.710, E3 +112617.351}
SPL {X  -148.063, Y  +312.768, Z    +0.000, E1   +70.492, E3 +112626.672}
SPL {X  -143.809, Y  +304.150, Z    +0.000, E1   +70.034, E3 +112635.815}
SPL {X  -139.938, Y  +297.268, Z    +0.000, E1   +69.438, E3 +112644.405}
SPL {X  -136.192, Y  +291.270, Z    +0.000, E1   +68.926, E3 +112651.553}
SPL {X  -132.794, Y  +286.287, Z    +0.000, E1   +68.653, E3 +112656.347}
SPL {X  -129.555, Y  +281.880, Z    +0.000, E1   +68.043, E3 +112662.447}
SPL {X  -126.523, Y  +278.020, Z    +0.000, E1   +67.371, E3 +112667.938}
SPL {X  -119.204, Y  +269.591, Z    +0.000, E1   +69.726, E3 +112663.822}
SPL {X   -73.382, Y  +235.154, Z    +0.000, E1   +54.977, E3 +112829.499}
ENDSPLINE

SPLINE
SPL {X  -133.875, Y  +287.830, Z    +0.000, E1   +51.751, E3 +112968.701}
SPL {X  -153.240, Y  +325.474, Z    +0.000, E1   +39.999, E3 +112979.904}
SPL {X  -160.567, Y  +353.506, Z    +0.000, E1   +24.043, E3 +112980.398}
SPL {X  -162.437, Y  +369.334, Z    +0.000, E1   +11.998, E3 +112981.524}
SPL {X  -162.814, Y  +379.161, Z    +0.000, E1    +3.343, E3 +112981.544}
SPL {X  -162.820, Y  +382.500, Z    +0.000, E1    +0.000, E3 +112981.026}
SPL {X  -162.820, Y  +384.390, Z    +0.000, E1    -3.279, E3 +112980.744}
SPL {X  -162.820, Y  +388.496, Z    +0.000, E1   -11.991, E3 +112980.645}
SPL {X  -162.820, Y  +392.944, Z    +0.000, E1   -22.020, E3 +112980.670}
SPL {X  -162.820, Y  +397.954, Z    +0.000, E1   -32.843, E3 +112980.710}
SPL {X  -162.820, Y  +404.232, Z    +0.000, E1   -44.157, E3 +112980.718}
SPL {X  -162.820, Y  +415.904, Z    +0.000, E1   -58.030, E3 +112980.992}
SPL {X  -162.820, Y  +472.155, Z    +0.000, E1   -74.123, E3 +112991.095}
SPL {X  -162.820, Y  +654.572, Z    +0.000, E1   -72.288, E3 +113093.320}
SPL {X  -162.820, Y  +673.151, Z    +0.000, E1   -71.906, E3 +113109.889}
SPL {X  -161.514, Y  +694.081, Z    +0.000, E1   -71.845, E3 +113124.544}
SPL {X  -159.782, Y  +704.807, Z    +0.000, E1   -71.464, E3 +113135.527}
SPL {X  -157.050, Y  +716.463, Z    +0.000, E1   -71.316, E3 +113144.827}
SPL {X  -154.424, Y  +725.109, Z    +0.000, E1   -70.982, E3 +113153.678}
SPL {X  -151.195, Y  +733.918, Z    +0.000, E1   -70.611, E3 +113162.801}
SPL {X  -147.776, Y  +741.856, Z    +0.000, E1   -70.224, E3 +113171.249}
SPL {X  -143.411, Y  +750.594, Z    +0.000, E1   -69.653, E3 +113181.405}
SPL {X  -140.107, Y  +756.448, Z    +0.000, E1   -69.170, E3 +113188.421}
SPL {X  -136.484, Y  +762.283, Z    +0.000, E1   -68.639, E3 +113195.810}
SPL {X  -132.373, Y  +768.304, Z    +0.000, E1   -68.109, E3 +113202.680}
SPL {X  -129.138, Y  +772.665, Z    +0.000, E1   -67.631, E3 +113208.027}
SPL {X  -125.533, Y  +777.190, Z    +0.000, E1   -67.475, E3 +113211.725}
SPL {X   -73.826, Y  +818.621, Z    +0.000, E1   -58.574, E3 +113307.218}
ENDSPLINE

SPLINE
SPL {X  -110.901, Y  +792.711, Z    +0.000, E1   -55.300, E3 +113492.076}
SPL {X  -144.508, Y  +748.519, Z    +0.000, E1   -46.961, E3 +113517.112}
SPL {X  -158.446, Y  +710.986, Z    +0.000, E1   -30.228, E3 +113520.477}
SPL {X  -162.035, Y  +689.470, Z    +0.000, E1   -15.657, E3 +113522.048}
SPL {X  -162.696, Y  +679.865, Z    +0.000, E1    -7.693, E3 +113522.120}
SPL {X  -162.820, Y  +671.472, Z    +0.000, E1    -0.171, E3 +113521.459}
SPL {X  -162.820, Y  +667.499, Z    +0.000, E1    +7.374, E3 +113521.200}
SPL {X  -162.820, Y  +663.777, Z    +0.000, E1   +15.496, E3 +113521.063}
SPL {X  -162.820, Y  +659.610, Z    +0.000, E1   +24.615, E3 +113521.108}
SPL {X  -162.820, Y  +654.471, Z    +0.000, E1   +35.284, E3 +113521.010}
SPL {X  -162.820, Y  +648.111, Z    +0.000, E1   +44.823, E3 +113522.308}
SPL {X  -162.820, Y  +635.984, Z    +0.000, E1   +61.208, E3 +113519.316}
SPL {X  -162.820, Y  +617.261, Z    +0.000, E1   +67.803, E3 +113524.502}
SPL {X  -162.820, Y  +579.681, Z    +0.000, E1   +72.301, E3 +113536.107}
SPL {X  -162.820, Y  +408.049, Z    +0.000, E1   +72.202, E3 +113628.539}
ENDSPLINE

SPLINE
SPL {X  -162.820, Y  +452.249, Z    +0.000, E1   +66.666, E3 +113644.545}
ENDSPLINE

SPLINE
SPL {X  -162.820, Y  +427.408, Z    +0.000, E1   +67.534, E3 +113659.163}
SPL {X  -162.820, Y  +402.068, Z    +0.000, E1   +68.403, E3 +113673.224}
SPL {X  -162.804, Y  +378.229, Z    +0.000, E1   +69.183, E3 +113685.551}
SPL {X  -161.511, Y  +359.895, Z    +0.000, E1   +69.744, E3 +113694.843}
SPL {X  -158.246, Y  +342.178, Z    +0.000, E1   +70.136, E3 +113704.592}
SPL {X  -152.677, Y  +323.931, Z    +0.000, E1   +70.710, E3 +113712.589}
SPL {X  -148.063, Y  +312.768, Z    +0.000, E1   +70.492, E3 +113721.910}
SPL {X  -143.809, Y  +304.150, Z    +0.000, E1   +70.034, E3 +113731.053}
SPL {X  -139.938, Y  +297.268, Z    +0.000, E1   +69.438, E3 +113739.644}
SPL {X  -136.192, Y  +291.270, Z    +0.000, E1   +68.926, E3 +113746.791}
SPL {X  -131.963, Y  +285.127, Z    +0.000, E1   +68.405, E3 +113753.781}
SPL {X  -127.466, Y  +279.195, Z    +0.000, E1   +67.714, E3 +113761.069}
SPL {X  -119.204, Y  +269.591, Z    +0.000, E1   +69.726, E3 +113759.060}
SPL {X   -73.382, Y  +235.154, Z    +0.000, E1   +54.977, E3 +113924.737}
ENDSPLINE

SPLINE
SPL {X  -133.875, Y  +287.830, Z    +0.000, E1   +51.751, E3 +114063.939}
SPL {X  -153.240, Y  +325.474, Z    +0.000, E1   +39.999, E3 +114075.142}
SPL {X  -159.032, Y  +345.583, Z    +0.000, E1   +29.156, E3 +114075.627}
SPL {X  -161.304, Y  +358.334, Z    +0.000, E1   +20.524, E3 +114075.584}
SPL {X  -162.437, Y  +369.334, Z    +0.000, E1   +11.998, E3 +114076.763}
SPL {X  -162.814, Y  +379.161, Z    +0.000, E1    +3.343, E3 +114076.782}
SPL {X  -162.820, Y  +382.500, Z    +0.000, E1    +0.000, E3 +114076.264}
SPL {X  -162.820, Y  +384.390, Z    +0.000, E1    -3.279, E3 +114075.982}
SPL {X  -162.820, Y  +388.496, Z    +0.000, E1   -11.991, E3 +114075.883}
SPL {X  -162.820, Y  +392.944, Z    +0.000, E1   -22.020, E3 +114075.908}
SPL {X  -162.820, Y  +397.954, Z    +0.000, E1   -32.843, E3 +114075.948}
SPL {X  -162.820, Y  +404.232, Z    +0.000, E1   -44.157, E3 +114075.956}
SPL {X  -162.820, Y  +415.904, Z    +0.000, E1   -58.030, E3 +114076.230}
SPL {X  -162.820, Y  +472.155, Z    +0.000, E1   -74.123, E3 +114086.333}
SPL {X  -162.820, Y  +661.743, Z    +0.000, E1   -73.395, E3 +114181.467}
ENDSPLINE

SPLINE
SPL {X  -162.820, Y  +658.105, Z    +0.000, E1   -71.889, E3 +114194.865}
ENDSPLINE

SPLINE
SPL {X  -162.784, Y  +676.927, Z    +0.000, E1   -71.815, E3 +114208.393}
SPL {X  -161.514, Y  +694.081, Z    +0.000, E1   -71.845, E3 +114219.782}
SPL {X  -159.782, Y  +704.807, Z    +0.000, E1   -71.464, E3 +114230.765}
SPL {X  -157.050, Y  +716.463, Z    +0.000, E1   -71.316, E3 +114240.065}
SPL {X  -154.424, Y  +725.109, Z    +0.000, E1   -70.982, E3 +114248.917}
SPL {X  -151.195, Y  +733.918, Z    +0.000, E1   -70.611, E3 +114258.039}
SPL {X  -147.776, Y  +741.856, Z    +0.000, E1   -70.224, E3 +114266.487}
SPL {X  -144.623, Y  +748.297, Z    +0.000, E1   -69.772, E3 +114274.112}
SPL {X  -141.153, Y  +754.655, Z    +0.000, E1   -69.344, E3 +114281.415}
SPL {X  -137.365, Y  +760.914, Z    +0.000, E1   -68.751, E3 +114289.354}
SPL {X  -133.334, Y  +766.947, Z    +0.000, E1   -68.226, E3 +114296.458}
SPL {X  -129.138, Y  +772.665, Z    +0.000, E1   -67.631, E3 +114303.265}
SPL {X  -125.533, Y  +777.190, Z    +0.000, E1   -67.475, E3 +114306.963}
SPL {X   -73.826, Y  +818.621, Z    +0.000, E1   -58.574, E3 +114402.456}
ENDSPLINE

SPLINE
SPL {X  -110.901, Y  +792.711, Z    +0.000, E1   -55.300, E3 +114587.314}
SPL {X  -144.508, Y  +748.519, Z    +0.000, E1   -46.961, E3 +114612.350}
SPL {X  -158.446, Y  +710.986, Z    +0.000, E1   -30.228, E3 +114615.715}
SPL {X  -162.035, Y  +689.470, Z    +0.000, E1   -15.657, E3 +114617.286}
SPL {X  -162.788, Y  +676.746, Z    +0.000, E1    -5.020, E3 +114617.194}
SPL {X  -162.820, Y  +671.525, Z    +0.000, E1    -0.042, E3 +114616.748}
SPL {X  -162.820, Y  +669.531, Z    +0.000, E1    +3.299, E3 +114616.437}
SPL {X  -162.820, Y  +664.807, Z    +0.000, E1   +13.064, E3 +114616.365}
SPL {X  -162.820, Y  +659.610, Z    +0.000, E1   +24.615, E3 +114616.346}
SPL {X  -162.820, Y  +651.281, Z    +0.000, E1   +40.220, E3 +114616.899}
SPL {X  -162.820, Y  +632.362, Z    +0.000, E1   +62.930, E3 +114615.559}
SPL {X  -162.820, Y  +579.681, Z    +0.000, E1   +72.301, E3 +114631.345}
SPL {X  -162.820, Y  +408.049, Z    +0.000, E1   +72.202, E3 +114723.777}
ENDSPLINE

SPLINE
SPL {X  -162.820, Y  +452.249, Z    +0.000, E1   +66.666, E3 +114739.783}
ENDSPLINE

SPLINE
SPL {X  -162.820, Y  +427.408, Z    +0.000, E1   +67.534, E3 +114754.401}
SPL {X  -162.820, Y  +409.075, Z    +0.000, E1   +68.145, E3 +114764.786}
SPL {X  -162.820, Y  +384.968, Z    +0.000, E1   +68.973, E3 +114777.345}
SPL {X  -162.073, Y  +364.922, Z    +0.000, E1   +69.599, E3 +114787.470}
SPL {X  -158.958, Y  +345.247, Z    +0.000, E1   +70.087, E3 +114798.066}
SPL {X  -154.257, Y  +328.393, Z    +0.000, E1   +70.602, E3 +114805.623}
SPL {X  -151.417, Y  +320.641, Z    +0.000, E1   +70.773, E3 +114809.506}
SPL {X  -148.063, Y  +312.768, Z    +0.000, E1   +70.492, E3 +114817.149}
SPL {X  -143.809, Y  +304.150, Z    +0.000, E1   +70.034, E3 +114826.291}
SPL {X  -139.938, Y  +297.268, Z    +0.000, E1   +69.438, E3 +114834.882}
SPL {X  -136.192, Y  +291.270, Z    +0.000, E1   +68.926, E3 +114842.029}
SPL {X  -131.963, Y  +285.127, Z    +0.000, E1   +68.405, E3 +114849.019}
SPL {X  -127.466, Y  +279.195, Z    +0.000, E1   +67.714, E3 +114856.307}
SPL {X  -119.204, Y  +269.591, Z    +0.000, E1   +69.726, E3 +114854.298}
SPL {X   -73.382, Y  +235.154, Z    +0.000, E1   +54.977, E3 +115019.975}
ENDSPLINE

SPLINE
SPL {X  -133.875, Y  +287.830, Z    +0.000, E1   +51.751, E3 +115159.177}
SPL {X  -153.240, Y  +325.474, Z    +0.000, E1   +39.999, E3 +115170.381}
SPL {X  -160.567, Y  +353.506, Z    +0.000, E1   +24.043, E3 +115170.875}
SPL {X  -162.646, Y  +372.968, Z    +0.000, E1    +8.995, E3 +115172.051}
SPL {X  -162.820, Y  +382.382, Z    +0.000, E1    +0.204, E3 +115171.538}
SPL {X  -162.820, Y  +384.390, Z    +0.000, E1    -3.279, E3 +115171.220}
SPL {X  -162.820, Y  +388.496, Z    +0.000, E1   -11.991, E3 +115171.121}
SPL {X  -162.820, Y  +392.944, Z    +0.000, E1   -22.020, E3 +115171.146}
SPL {X  -162.820, Y  +397.954, Z    +0.000, E1   -32.843, E3 +115171.186}
SPL {X  -162.820, Y  +404.232, Z    +0.000, E1   -44.157, E3 +115171.195}
SPL {X  -162.820, Y  +415.904, Z    +0.000, E1   -58.030, E3 +115171.468}
SPL {X  -162.820, Y  +472.155, Z    +0.000, E1   -74.123, E3 +115181.571}
SPL {X  -162.820, Y  +661.743, Z    +0.000, E1   -73.395, E3 +115276.705}
ENDSPLINE

SPLINE
SPL {X  -162.820, Y  +658.105, Z    +0.000, E1   -71.889, E3 +115290.103}
ENDSPLINE

SPLINE
SPL {X  -162.784, Y  +676.927, Z    +0.000, E1   -71.815, E3 +115303.631}
SPL {X  -161.514, Y  +694.081, Z    +0.000, E1   -71.845, E3 +115315.021}
SPL {X  -159.782, Y  +704.807, Z    +0.000, E1   -71.464, E3 +115326.003}
SPL {X  -157.050, Y  +716.463, Z    +0.000, E1   -71.316, E3 +115335.303}
SPL {X  -154.424, Y  +725.109, Z    +0.000, E1   -70.982, E3 +115344.155}
SPL {X  -151.195, Y  +733.918, Z    +0.000, E1   -70.611, E3 +115353.277}
SPL {X  -147.776, Y  +741.856, Z    +0.000, E1   -70.224, E3 +115361.725}
SPL {X  -143.411, Y  +750.594, Z    +0.000, E1   -69.653, E3 +115371.881}
SPL {X  -138.205, Y  +759.580, Z    +0.000, E1   -68.913, E3 +115382.830}
SPL {X  -133.334, Y  +766.947, Z    +0.000, E1   -68.226, E3 +115391.696}
SPL {X  -129.138, Y  +772.665, Z    +0.000, E1   -67.631, E3 +115398.503}
SPL {X  -125.533, Y  +777.190, Z    +0.000, E1   -67.475, E3 +115402.201}
SPL {X   -75.773, Y  +817.614, Z    +0.000, E1   -59.878, E3 +115483.166}
SPL {X   -71.637, Y  +819.714, Z    +0.000, E1   -56.371, E3 +115528.773}
ENDSPLINE

SPLINE
SPL {X  -110.901, Y  +792.711, Z    +0.000, E1   -55.300, E3 +115682.552}
SPL {X  -144.508, Y  +748.519, Z    +0.000, E1   -46.961, E3 +115707.588}
SPL {X  -156.638, Y  +717.940, Z    +0.000, E1   -34.002, E3 +115710.324}
SPL {X  -160.830, Y  +698.875, Z    +0.000, E1   -22.517, E3 +115711.988}
SPL {X  -162.532, Y  +683.174, Z    +0.000, E1   -10.600, E3 +115712.593}
SPL {X  -162.820, Y  +671.754, Z    +0.000, E1    -0.424, E3 +115712.010}
SPL {X  -162.820, Y  +670.529, Z    +0.000, E1    +1.628, E3 +115711.688}
SPL {X  -162.820, Y  +667.499, Z    +0.000, E1    +7.374, E3 +115711.676}
SPL {X  -162.820, Y  +663.777, Z    +0.000, E1   +15.496, E3 +115711.539}
SPL {X  -162.820, Y  +659.610, Z    +0.000, E1   +24.615, E3 +115711.584}
SPL {X  -162.820, Y  +651.281, Z    +0.000, E1   +40.220, E3 +115712.137}
SPL {X  -162.820, Y  +632.362, Z    +0.000, E1   +62.930, E3 +115710.797}
SPL {X  -162.820, Y  +579.681, Z    +0.000, E1   +72.301, E3 +115726.583}
SPL {X  -162.820, Y  +408.049, Z    +0.000, E1   +72.202, E3 +115819.015}
ENDSPLINE

SPLINE
SPL {X  -162.820, Y  +452.249, Z    +0.000, E1   +66.666, E3 +115835.021}
ENDSPLINE

SPLINE
SPL {X  -162.820, Y  +427.408, Z    +0.000, E1   +67.534, E3 +115849.639}
SPL {X  -162.820, Y  +402.068, Z    +0.000, E1   +68.403, E3 +115863.701}
SPL {X  -162.804, Y  +378.229, Z    +0.000, E1   +69.183, E3 +115876.028}
SPL {X  -161.511, Y  +359.895, Z    +0.000, E1   +69.744, E3 +115885.319}
SPL {X  -158.246, Y  +342.178, Z    +0.000, E1   +70.136, E3 +115895.069}
SPL {X  -154.257, Y  +328.393, Z    +0.000, E1   +70.602, E3 +115900.861}
SPL {X  -150.447, Y  +318.243, Z    +0.000, E1   +70.683, E3 +115907.208}
SPL {X  -145.895, Y  +308.216, Z    +0.000, E1   +70.273, E3 +115917.161}
SPL {X  -140.654, Y  +298.483, Z    +0.000, E1   +69.615, E3 +115928.303}
SPL {X  -136.192, Y  +291.270, Z    +0.000, E1   +68.926, E3 +115937.267}
SPL {X  -132.794, Y  +286.287, Z    +0.000, E1   +68.653, E3 +115942.062}
SPL {X  -129.555, Y  +281.880, Z    +0.000, E1   +68.043, E3 +115948.162}
SPL {X  -126.523, Y  +278.020, Z    +0.000, E1   +67.371, E3 +115953.653}
SPL {X  -119.204, Y  +269.591, Z    +0.000, E1   +69.726, E3 +115949.536}
SPL {X   -73.382, Y  +235.154, Z    +0.000, E1   +54.977, E3 +116115.213}
ENDSPLINE

SPLINE
SPL {X  -115.538, Y  +265.778, Z    +0.000, E1   +55.826, E3 +116245.664}
SPL {X  -140.740, Y  +298.630, Z    +0.000, E1   +48.901, E3 +116256.999}
SPL {X  -153.240, Y  +325.474, Z    +0.000, E1   +39.999, E3 +116265.619}
SPL {X  -160.567, Y  +353.506, Z    +0.000, E1   +24.043, E3 +116266.113}
SPL {X  -162.437, Y  +369.334, Z    +0.000, E1   +11.998, E3 +116267.239}
SPL {X  -162.814, Y  +379.161, Z    +0.000, E1    +3.343, E3 +116267.258}
SPL {X  -162.820, Y  +382.500, Z    +0.000, E1    +0.000, E3 +116266.741}
SPL {X  -162.820, Y  +384.390, Z    +0.000, E1    -3.279, E3 +116266.458}
SPL {X  -162.820, Y  +388.496, Z    +0.000, E1   -11.991, E3 +116266.360}
SPL {X  -162.820, Y  +392.944, Z    +0.000, E1   -22.020, E3 +116266.384}
SPL {X  -162.820, Y  +397.954, Z    +0.000, E1   -32.843, E3 +116266.425}
SPL {X  -162.820, Y  +404.232, Z    +0.000, E1   -44.157, E3 +116266.433}
SPL {X  -162.820, Y  +415.904, Z    +0.000, E1   -58.030, E3 +116266.706}
SPL {X  -162.820, Y  +472.155, Z    +0.000, E1   -74.123, E3 +116276.809}
SPL {X  -162.820, Y  +661.743, Z    +0.000, E1   -73.395, E3 +116371.943}
ENDSPLINE

SPLINE
SPL {X  -162.820, Y  +658.105, Z    +0.000, E1   -71.889, E3 +116385.341}
ENDSPLINE

SPLINE
SPL {X  -162.784, Y  +676.927, Z    +0.000, E1   -71.815, E3 +116398.869}
SPL {X  -161.514, Y  +694.081, Z    +0.000, E1   -71.845, E3 +116410.259}
SPL {X  -159.782, Y  +704.807, Z    +0.000, E1   -71.464, E3 +116421.241}
SPL {X  -157.050, Y  +716.463, Z    +0.000, E1   -71.316, E3 +116430.541}
SPL {X  -154.424, Y  +725.109, Z    +0.000, E1   -70.982, E3 +116439.393}
SPL {X  -151.195, Y  +733.918, Z    +0.000, E1   -70.611, E3 +116448.515}
SPL {X  -147.776, Y  +741.856, Z    +0.000, E1   -70.224, E3 +116456.963}
SPL {X  -143.411, Y  +750.594, Z    +0.000, E1   -69.653, E3 +116467.119}
SPL {X  -140.107, Y  +756.448, Z    +0.000, E1   -69.170, E3 +116474.135}
SPL {X  -136.484, Y  +762.283, Z    +0.000, E1   -68.639, E3 +116481.524}
SPL {X  -131.125, Y  +770.022, Z    +0.000, E1   -67.959, E3 +116490.431}
SPL {X  -126.438, Y  +776.086, Z    +0.000, E1   -67.465, E3 +116496.753}
SPL {X   -73.826, Y  +818.621, Z    +0.000, E1   -58.574, E3 +116592.932}
ENDSPLINE

SPLINE
SPL {X  -110.901, Y  +792.711, Z    +0.000, E1   -55.300, E3 +116777.790}
SPL {X  -144.508, Y  +748.519, Z    +0.000, E1   -46.961, E3 +116802.826}
SPL {X  -158.446, Y  +710.986, Z    +0.000, E1   -30.228, E3 +116806.191}
SPL {X  -162.035, Y  +689.470, Z    +0.000, E1   -15.657, E3 +116807.762}
SPL {X  -162.696, Y  +679.865, Z    +0.000, E1    -7.693, E3 +116807.834}
SPL {X  -162.820, Y  +671.754, Z    +0.000, E1    -0.424, E3 +116807.248}
SPL {X  -162.820, Y  +669.531, Z    +0.000, E1    +3.299, E3 +116806.913}
SPL {X  -162.820, Y  +664.807, Z    +0.000, E1   +13.064, E3 +116806.842}
SPL {X  -162.820, Y  +659.610, Z    +0.000, E1   +24.615, E3 +116806.823}
SPL {X  -162.820, Y  +654.471, Z    +0.000, E1   +35.284, E3 +116806.725}
SPL {X  -162.820, Y  +648.111, Z    +0.000, E1   +44.823, E3 +116808.022}
SPL {X  -162.820, Y  +632.362, Z    +0.000, E1   +62.930, E3 +116806.035}
SPL {X  -162.820, Y  +579.681, Z    +0.000, E1   +72.301, E3 +116821.821}
SPL {X  -162.820, Y  +402.073, Z    +0.000, E1   +73.274, E3 +116907.356}
ENDSPLINE

SPLINE
SPL {X  -162.820, Y  +412.258, Z    +0.000, E1   +71.454, E3 +116918.453}
SPL {X  -162.820, Y  +452.249, Z    +0.000, E1   +66.666, E3 +116930.259}
ENDSPLINE

SPLINE
SPL {X  -162.820, Y  +427.408, Z    +0.000, E1   +67.534, E3 +116944.877}
SPL {X  -162.820, Y  +402.068, Z    +0.000, E1   +68.403, E3 +116958.939}
SPL {X  -162.804, Y  +378.229, Z    +0.000, E1   +69.183, E3 +116971.266}
SPL {X  -161.511, Y  +359.895, Z    +0.000, E1   +69.744, E3 +116980.557}
SPL {X  -158.246, Y  +342.178, Z    +0.000, E1   +70.136, E3 +116990.307}
SPL {X  -154.257, Y  +328.393, Z    +0.000, E1   +70.602, E3 +116996.099}
SPL {X  -151.417, Y  +320.641, Z    +0.000, E1   +70.773, E3 +116999.982}
SPL {X  -148.063, Y  +312.768, Z    +0.000, E1   +70.492, E3 +117007.625}
SPL {X  -143.809, Y  +304.150, Z    +0.000, E1   +70.034, E3 +117016.767}
SPL {X  -139.938, Y  +297.268, Z    +0.000, E1   +69.438, E3 +117025.358}
SPL {X  -136.192, Y  +291.270, Z    +0.000, E1   +68.926, E3 +117032.505}
SPL {X  -131.963, Y  +285.127, Z    +0.000, E1   +68.405, E3 +117039.495}
SPL {X  -127.466, Y  +279.195, Z    +0.000, E1   +67.714, E3 +117046.783}
SPL {X  -119.204, Y  +269.591, Z    +0.000, E1   +69.726, E3 +117044.774}
SPL {X   -73.382, Y  +235.154, Z    +0.000, E1   +54.977, E3 +117210.451}
ENDSPLINE

SPLINE
SPL {X  -133.875, Y  +287.830, Z    +0.000, E1   +51.751, E3 +117349.653}
SPL {X  -153.240, Y  +325.474, Z    +0.000, E1   +39.999, E3 +117360.857}
SPL {X  -160.567, Y  +353.506, Z    +0.000, E1   +24.043, E3 +117361.351}
SPL {X  -162.646, Y  +372.968, Z    +0.000, E1    +8.995, E3 +117362.528}
SPL {X  -162.820, Y  +382.382, Z    +0.000, E1    +0.204, E3 +117362.015}
SPL {X  -162.820, Y  +384.390, Z    +0.000, E1    -3.279, E3 +117361.696}
SPL {X  -162.820, Y  +388.496, Z    +0.000, E1   -11.991, E3 +117361.598}
SPL {X  -162.820, Y  +392.944, Z    +0.000, E1   -22.020, E3 +117361.622}
SPL {X  -162.820, Y  +397.954, Z    +0.000, E1   -32.843, E3 +117361.663}
SPL {X  -162.820, Y  +404.232, Z    +0.000, E1   -44.157, E3 +117361.671}
SPL {X  -162.820, Y  +415.904, Z    +0.000, E1   -58.030, E3 +117361.944}
SPL {X  -162.820, Y  +467.484, Z    +0.000, E1   -73.355, E3 +117371.774}
SPL {X  -162.820, Y  +491.822, Z    +0.000, E1   -76.748, E3 +117373.197}
SPL {X  -162.820, Y  +654.572, Z    +0.000, E1   -72.288, E3 +117474.273}
SPL {X  -162.820, Y  +673.151, Z    +0.000, E1   -71.906, E3 +117490.842}
SPL {X  -161.514, Y  +694.081, Z    +0.000, E1   -71.845, E3 +117505.497}
SPL {X  -159.782, Y  +704.807, Z    +0.000, E1   -71.464, E3 +117516.479}
SPL {X  -157.050, Y  +716.463, Z    +0.000, E1   -71.316, E3 +117525.779}
SPL {X  -154.424, Y  +725.109, Z    +0.000, E1   -70.982, E3 +117534.631}
SPL {X  -151.195, Y  +733.918, Z    +0.000, E1   -70.611, E3 +117543.753}
SPL {X  -147.776, Y  +741.856, Z    +0.000, E1   -70.224, E3 +117552.201}
SPL {X  -143.411, Y  +750.594, Z    +0.000, E1   -69.653, E3 +117562.357}
SPL {X  -138.205, Y  +759.580, Z    +0.000, E1   -68.913, E3 +117573.307}
SPL {X  -133.334, Y  +766.947, Z    +0.000, E1   -68.226, E3 +117582.173}
SPL {X  -129.138, Y  +772.665, Z    +0.000, E1   -67.631, E3 +117588.979}
SPL {X  -125.533, Y  +777.190, Z    +0.000, E1   -67.475, E3 +117592.677}
SPL {X   -73.826, Y  +818.621, Z    +0.000, E1   -58.574, E3 +117688.170}
ENDSPLINE

SPLINE
SPL {X  -110.901, Y  +792.711, Z    +0.000, E1   -55.300, E3 +117873.028}
SPL {X  -144.508, Y  +748.519, Z    +0.000, E1   -46.961, E3 +117898.064}
SPL {X  -156.638, Y  +717.940, Z    +0.000, E1   -34.002, E3 +117900.800}
SPL {X  -160.830, Y  +698.875, Z    +0.000, E1   -22.517, E3 +117902.464}
SPL {X  -162.532, Y  +683.174, Z    +0.000, E1   -10.600, E3 +117903.069}
SPL {X  -162.820, Y  +671.472, Z    +0.000, E1    -0.171, E3 +117902.412}
SPL {X  -162.820, Y  +667.499, Z    +0.000, E1    +7.374, E3 +117902.152}
SPL {X  -162.820, Y  +663.777, Z    +0.000, E1   +15.496, E3 +117902.015}
SPL {X  -162.820, Y  +659.610, Z    +0.000, E1   +24.615, E3 +117902.061}
SPL {X  -162.820, Y  +651.281, Z    +0.000, E1   +40.220, E3 +117902.614}
SPL {X  -162.820, Y  +632.362, Z    +0.000, E1   +62.930, E3 +117901.273}
SPL {X  -162.820, Y  +579.681, Z    +0.000, E1   +72.301, E3 +117917.059}
SPL {X  -162.820, Y  +408.049, Z    +0.000, E1   +72.202, E3 +118009.491}
ENDSPLINE

SPLINE
SPL {X  -162.820, Y  +452.249, Z    +0.000, E1   +66.666, E3 +118025.497}
ENDSPLINE

SPLINE
SPL {X  -162.820, Y  +427.408, Z    +0.000, E1   +67.534, E3 +118040.115}
SPL {X  -162.820, Y  +402.068, Z    +0.000, E1   +68.403, E3 +118054.177}
SPL {X  -162.523, Y  +370.677, Z    +0.000, E1   +69.437, E3 +118070.238}
SPL {X  -158.958, Y  +345.247, Z    +0.000, E1   +70.087, E3 +118083.780}
SPL {X  -152.677, Y  +323.931, Z    +0.000, E1   +70.710, E3 +118093.542}
SPL {X  -148.063, Y  +312.768, Z    +0.000, E1   +70.492, E3 +118102.863}
SPL {X  -143.809, Y  +304.150, Z    +0.000, E1   +70.034, E3 +118112.006}
SPL {X  -139.938, Y  +297.268, Z    +0.000, E1   +69.438, E3 +118120.596}
SPL {X  -136.192, Y  +291.270, Z    +0.000, E1   +68.926, E3 +118127.743}
SPL {X  -132.794, Y  +286.287, Z    +0.000, E1   +68.653, E3 +118132.538}
SPL {X  -129.555, Y  +281.880, Z    +0.000, E1   +68.043, E3 +118138.638}
SPL {X  -126.523, Y  +278.020, Z    +0.000, E1   +67.371, E3 +118144.129}
SPL {X  -119.204, Y  +269.591, Z    +0.000, E1   +69.726, E3 +118140.012}
SPL {X   -73.382, Y  +235.154, Z    +0.000, E1   +54.977, E3 +118305.689}
ENDSPLINE

SPLINE
SPL {X  -133.875, Y  +287.830, Z    +0.000, E1   +51.751, E3 +118444.892}
SPL {X  -153.240, Y  +325.474, Z    +0.000, E1   +39.999, E3 +118456.095}
SPL {X  -160.567, Y  +353.506, Z    +0.000, E1   +24.043, E3 +118456.589}
SPL {X  -162.437, Y  +369.334, Z    +0.000, E1   +11.998, E3 +118457.715}
SPL {X  -162.814, Y  +379.161, Z    +0.000, E1    +3.343, E3 +118457.734}
SPL {X  -162.820, Y  +382.751, Z    +0.000, E1    -0.252, E3 +118457.148}
SPL {X  -162.820, Y  +387.406, Z    +0.000, E1    -9.377, E3 +118456.869}
SPL {X  -162.820, Y  +392.944, Z    +0.000, E1   -22.020, E3 +118456.861}
SPL {X  -162.820, Y  +397.954, Z    +0.000, E1   -32.843, E3 +118456.901}
SPL {X  -162.820, Y  +404.232, Z    +0.000, E1   -44.157, E3 +118456.909}
SPL {X  -162.820, Y  +415.904, Z    +0.000, E1   -58.030, E3 +118457.182}
SPL {X  -162.820, Y  +467.484, Z    +0.000, E1   -73.355, E3 +118467.012}
SPL {X  -162.820, Y  +491.822, Z    +0.000, E1   -76.748, E3 +118468.435}
SPL {X  -162.820, Y  +661.743, Z    +0.000, E1   -73.395, E3 +118562.419}
ENDSPLINE

SPLINE
SPL {X  -162.820, Y  +658.105, Z    +0.000, E1   -71.889, E3 +118575.817}
ENDSPLINE

SPLINE
SPL {X  -162.784, Y  +676.927, Z    +0.000, E1   -71.815, E3 +118589.345}
SPL {X  -161.514, Y  +694.081, Z    +0.000, E1   -71.845, E3 +118600.735}
SPL {X  -159.782, Y  +704.807, Z    +0.000, E1   -71.464, E3 +118611.717}
SPL {X  -157.050, Y  +716.463, Z    +0.000, E1   -71.316, E3 +118621.017}
SPL {X  -154.424, Y  +725.109, Z    +0.000, E1   -70.982, E3 +118629.869}
SPL {X  -151.195, Y  +733.918, Z    +0.000, E1   -70.611, E3 +118638.991}
SPL {X  -147.776, Y  +741.856, Z    +0.000, E1   -70.224, E3 +118647.439}
SPL {X  -144.623, Y  +748.297, Z    +0.000, E1   -69.772, E3 +118655.064}
SPL {X  -141.153, Y  +754.655, Z    +0.000, E1   -69.344, E3 +118662.368}
SPL {X  -137.365, Y  +760.914, Z    +0.000, E1   -68.751, E3 +118670.306}
SPL {X  -133.334, Y  +766.947, Z    +0.000, E1   -68.226, E3 +118677.411}
SPL {X  -129.138, Y  +772.665, Z    +0.000, E1   -67.631, E3 +118684.218}
SPL {X  -125.533, Y  +777.190, Z    +0.000, E1   -67.475, E3 +118687.915}
SPL {X   -73.826, Y  +818.621, Z    +0.000, E1   -58.574, E3 +118783.408}
ENDSPLINE

SPLINE
SPL {X  -110.901, Y  +792.711, Z    +0.000, E1   -55.300, E3 +118968.266}
SPL {X  -144.508, Y  +748.519, Z    +0.000, E1   -46.961, E3 +118993.303}
SPL {X  -158.446, Y  +710.986, Z    +0.000, E1   -30.228, E3 +118996.668}
SPL {X  -162.035, Y  +689.470, Z    +0.000, E1   -15.657, E3 +118998.239}
SPL {X  -162.788, Y  +676.746, Z    +0.000, E1    -5.020, E3 +118998.146}
SPL {X  -162.820, Y  +671.525, Z    +0.000, E1    -0.042, E3 +118997.700}
SPL {X  -162.820, Y  +669.531, Z    +0.000, E1    +3.299, E3 +118997.389}
SPL {X  -162.820, Y  +664.807, Z    +0.000, E1   +13.064, E3 +118997.318}
SPL {X  -162.820, Y  +659.610, Z    +0.000, E1   +24.615, E3 +118997.299}
SPL {X  -162.820, Y  +651.281, Z    +0.000, E1   +40.220, E3 +118997.852}
SPL {X  -162.820, Y  +635.984, Z    +0.000, E1   +61.208, E3 +118995.506}
SPL {X  -162.820, Y  +617.261, Z    +0.000, E1   +67.803, E3 +119000.692}
SPL {X  -162.820, Y  +579.681, Z    +0.000, E1   +72.301, E3 +119012.297}
SPL {X  -162.820, Y  +408.049, Z    +0.000, E1   +72.202, E3 +119104.729}
ENDSPLINE

SPLINE
SPL {X  -162.820, Y  +452.249, Z    +0.000, E1   +66.666, E3 +119120.735}
ENDSPLINE

SPLINE
SPL {X  -162.820, Y  +427.408, Z    +0.000, E1   +67.534, E3 +119135.353}
SPL {X  -162.820, Y  +409.075, Z    +0.000, E1   +68.145, E3 +119145.738}
SPL {X  -162.820, Y  +384.968, Z    +0.000, E1   +68.973, E3 +119158.298}
SPL {X  -161.511, Y  +359.895, Z    +0.000, E1   +69.744, E3 +119171.034}
SPL {X  -158.246, Y  +342.178, Z    +0.000, E1   +70.136, E3 +119180.783}
SPL {X  -152.677, Y  +323.931, Z    +0.000, E1   +70.710, E3 +119188.780}
SPL {X  -148.063, Y  +312.768, Z    +0.000, E1   +70.492, E3 +119198.101}
SPL {X  -143.809, Y  +304.150, Z    +0.000, E1   +70.034, E3 +119207.244}
SPL {X  -139.938, Y  +297.268, Z    +0.000, E1   +69.438, E3 +119215.834}
SPL {X  -136.192, Y  +291.270, Z    +0.000, E1   +68.926, E3 +119222.981}
SPL {X  -132.794, Y  +286.287, Z    +0.000, E1   +68.653, E3 +119227.776}
SPL {X  -129.555, Y  +281.880, Z    +0.000, E1   +68.043, E3 +119233.876}
SPL {X  -126.523, Y  +278.020, Z    +0.000, E1   +67.371, E3 +119239.367}
SPL {X  -119.204, Y  +269.591, Z    +0.000, E1   +69.726, E3 +119235.250}
SPL {X   -73.382, Y  +235.154, Z    +0.000, E1   +54.977, E3 +119400.927}
ENDSPLINE

SPLINE
SPL {X  -133.875, Y  +287.830, Z    +0.000, E1   +51.751, E3 +119540.130}
SPL {X  -153.240, Y  +325.474, Z    +0.000, E1   +39.999, E3 +119551.333}
SPL {X  -159.032, Y  +345.583, Z    +0.000, E1   +29.156, E3 +119551.817}
SPL {X  -161.304, Y  +358.334, Z    +0.000, E1   +20.524, E3 +119551.774}
SPL {X  -162.646, Y  +372.968, Z    +0.000, E1    +8.995, E3 +119553.004}
SPL {X  -162.820, Y  +382.646, Z    +0.000, E1    -0.044, E3 +119552.418}
SPL {X  -162.820, Y  +387.406, Z    +0.000, E1    -9.377, E3 +119552.107}
SPL {X  -162.820, Y  +392.944, Z    +0.000, E1   -22.020, E3 +119552.099}
SPL {X  -162.820, Y  +397.954, Z    +0.000, E1   -32.843, E3 +119552.139}
SPL {X  -162.820, Y  +404.232, Z    +0.000, E1   -44.157, E3 +119552.147}
SPL {X  -162.820, Y  +415.904, Z    +0.000, E1   -58.030, E3 +119552.420}
SPL {X  -162.820, Y  +472.155, Z    +0.000, E1   -74.123, E3 +119562.523}
SPL {X  -162.820, Y  +654.572, Z    +0.000, E1   -72.288, E3 +119664.749}
SPL {X  -162.820, Y  +673.151, Z    +0.000, E1   -71.906, E3 +119681.318}
SPL {X  -161.514, Y  +694.081, Z    +0.000, E1   -71.845, E3 +119695.973}
SPL {X  -159.782, Y  +704.807, Z    +0.000, E1   -71.464, E3 +119706.955}
SPL {X  -157.050, Y  +716.463, Z    +0.000, E1   -71.316, E3 +119716.255}
SPL {X  -154.424, Y  +725.109, Z    +0.000, E1   -70.982, E3 +119725.107}
SPL {X  -151.195, Y  +733.918, Z    +0.000, E1   -70.611, E3 +119734.230}
SPL {X  -147.776, Y  +741.856, Z    +0.000, E1   -70.224, E3 +119742.678}
SPL {X  -144.623, Y  +748.297, Z    +0.000, E1   -69.772, E3 +119750.302}
SPL {X  -141.153, Y  +754.655, Z    +0.000, E1   -69.344, E3 +119757.606}
SPL {X  -136.484, Y  +762.283, Z    +0.000, E1   -68.639, E3 +119767.238}
SPL {X  -131.125, Y  +770.022, Z    +0.000, E1   -67.959, E3 +119776.145}
SPL {X  -126.438, Y  +776.086, Z    +0.000, E1   -67.465, E3 +119782.467}
SPL {X   -73.826, Y  +818.621, Z    +0.000, E1   -58.574, E3 +119878.646}
ENDSPLINE

SPLINE
SPL {X  -110.901, Y  +792.711, Z    +0.000, E1   -55.300, E3 +120063.504}
SPL {X  -144.508, Y  +748.519, Z    +0.000, E1   -46.961, E3 +120088.541}
SPL {X  -156.638, Y  +717.940, Z    +0.000, E1   -34.002, E3 +120091.276}
SPL {X  -160.830, Y  +698.875, Z    +0.000, E1   -22.517, E3 +120092.940}
SPL {X  -162.532, Y  +683.174, Z    +0.000, E1   -10.600, E3 +120093.546}
SPL {X  -162.820, Y  +671.472, Z    +0.000, E1    -0.171, E3 +120092.888}
SPL {X  -162.820, Y  +667.499, Z    +0.000, E1    +7.374, E3 +120092.629}
SPL {X  -162.820, Y  +663.777, Z    +0.000, E1   +15.496, E3 +120092.492}
SPL {X  -162.820, Y  +659.610, Z    +0.000, E1   +24.615, E3 +120092.537}
SPL {X  -162.820, Y  +654.471, Z    +0.000, E1   +35.284, E3 +120092.439}
SPL {X  -162.820, Y  +648.111, Z    +0.000, E1   +44.823, E3 +120093.736}
SPL {X  -162.820, Y  +635.984, Z    +0.000, E1   +61.208, E3 +120090.744}
SPL {X  -162.820, Y  +617.261, Z    +0.000, E1   +67.803, E3 +120095.931}
SPL {X  -162.820, Y  +579.681, Z    +0.000, E1   +72.301, E3 +120107.536}
SPL {X  -162.820, Y  +408.049, Z    +0.000, E1   +72.202, E3 +120199.967}
ENDSPLINE

SPLINE
SPL {X  -162.820, Y  +452.249, Z    +0.000, E1   +66.666, E3 +120215.973}
ENDSPLINE

SPLINE
SPL {X  -162.820, Y  +427.408, Z    +0.000, E1   +67.534, E3 +120230.592}
SPL {X  -162.820, Y  +402.068, Z    +0.000, E1   +68.403, E3 +120244.653}
SPL {X  -162.804, Y  +378.229, Z    +0.000, E1   +69.183, E3 +120256.980}
SPL {X  -161.511, Y  +359.895, Z    +0.000, E1   +69.744, E3 +120266.272}
SPL {X  -158.246, Y  +342.178, Z    +0.000, E1   +70.136, E3 +120276.021}
SPL {X  -154.257, Y  +328.393, Z    +0.000, E1   +70.602, E3 +120281.813}
SPL {X  -151.417, Y  +320.641, Z    +0.000, E1   +70.773, E3 +120285.697}
SPL {X  -148.063, Y  +312.768, Z    +0.000, E1   +70.492, E3 +120293.339}
SPL {X  -143.809, Y  +304.150, Z    +0.000, E1   +70.034, E3 +120302.482}
SPL {X  -139.938, Y  +297.268, Z    +0.000, E1   +69.438, E3 +120311.072}
SPL {X  -136.192, Y  +291.270, Z    +0.000, E1   +68.926, E3 +120318.219}
SPL {X  -131.963, Y  +285.127, Z    +0.000, E1   +68.405, E3 +120325.210}
SPL {X  -127.466, Y  +279.195, Z    +0.000, E1   +67.714, E3 +120332.497}
SPL {X  -119.204, Y  +269.591, Z    +0.000, E1   +69.726, E3 +120330.488}
SPL {X   -73.382, Y  +235.154, Z    +0.000, E1   +54.977, E3 +120496.165}
ENDSPLINE

SPLINE
SPL {X  -133.875, Y  +287.830, Z    +0.000, E1   +51.751, E3 +120635.368}
SPL {X  -153.240, Y  +325.474, Z    +0.000, E1   +39.999, E3 +120646.571}
SPL {X  -159.032, Y  +345.583, Z    +0.000, E1   +29.156, E3 +120647.055}
SPL {X  -161.304, Y  +358.334, Z    +0.000, E1   +20.524, E3 +120647.012}
SPL {X  -162.437, Y  +369.334, Z    +0.000, E1   +11.998, E3 +120648.191}
SPL {X  -162.814, Y  +379.161, Z    +0.000, E1    +3.343, E3 +120648.210}
SPL {X  -162.820, Y  +382.751, Z    +0.000, E1    -0.252, E3 +120647.624}
SPL {X  -162.820, Y  +387.406, Z    +0.000, E1    -9.377, E3 +120647.346}
SPL {X  -162.820, Y  +392.944, Z    +0.000, E1   -22.020, E3 +120647.337}
SPL {X  -162.820, Y  +397.954, Z    +0.000, E1   -32.843, E3 +120647.377}
SPL {X  -162.820, Y  +404.232, Z    +0.000, E1   -44.157, E3 +120647.385}
SPL {X  -162.820, Y  +415.904, Z    +0.000, E1   -58.030, E3 +120647.658}
SPL {X  -162.820, Y  +472.155, Z    +0.000, E1   -74.123, E3 +120657.761}
SPL {X  -162.820, Y  +654.572, Z    +0.000, E1   -72.288, E3 +120759.987}
SPL {X  -162.820, Y  +673.151, Z    +0.000, E1   -71.906, E3 +120776.556}
SPL {X  -161.514, Y  +694.081, Z    +0.000, E1   -71.845, E3 +120791.211}
SPL {X  -159.782, Y  +704.807, Z    +0.000, E1   -71.464, E3 +120802.193}
SPL {X  -157.050, Y  +716.463, Z    +0.000, E1   -71.316, E3 +120811.493}
SPL {X  -154.424, Y  +725.109, Z    +0.000, E1   -70.982, E3 +120820.345}
SPL {X  -151.195, Y  +733.918, Z    +0.000, E1   -70.611, E3 +120829.468}
SPL {X  -147.776, Y  +741.856, Z    +0.000, E1   -70.224, E3 +120837.916}
SPL {X  -144.623, Y  +748.297, Z    +0.000, E1   -69.772, E3 +120845.540}
SPL {X  -141.153, Y  +754.655, Z    +0.000, E1   -69.344, E3 +120852.844}
SPL {X  -137.365, Y  +760.914, Z    +0.000, E1   -68.751, E3 +120860.782}
SPL {X  -133.334, Y  +766.947, Z    +0.000, E1   -68.226, E3 +120867.887}
SPL {X  -129.138, Y  +772.665, Z    +0.000, E1   -67.631, E3 +120874.694}
SPL {X  -125.533, Y  +777.190, Z    +0.000, E1   -67.475, E3 +120878.391}
SPL {X   -73.826, Y  +818.621, Z    +0.000, E1   -58.574, E3 +120973.884}
ENDSPLINE

SPLINE
SPL {X  -110.901, Y  +792.711, Z    +0.000, E1   -55.300, E3 +121158.742}
SPL {X  -144.508, Y  +748.519, Z    +0.000, E1   -46.961, E3 +121183.779}
SPL {X  -156.638, Y  +717.940, Z    +0.000, E1   -34.002, E3 +121186.514}
SPL {X  -160.830, Y  +698.875, Z    +0.000, E1   -22.517, E3 +121188.178}
SPL {X  -162.277, Y  +686.786, Z    +0.000, E1   -13.481, E3 +121188.757}
SPL {X  -162.788, Y  +676.746, Z    +0.000, E1    -5.020, E3 +121188.622}
SPL {X  -162.820, Y  +671.525, Z    +0.000, E1    -0.042, E3 +121188.176}
SPL {X  -162.820, Y  +670.529, Z    +0.000, E1    +1.628, E3 +121187.878}
SPL {X  -162.820, Y  +667.499, Z    +0.000, E1    +7.374, E3 +121187.867}
SPL {X  -162.820, Y  +663.777, Z    +0.000, E1   +15.496, E3 +121187.730}
SPL {X  -162.820, Y  +659.610, Z    +0.000, E1   +24.615, E3 +121187.775}
SPL {X  -162.820, Y  +651.281, Z    +0.000, E1   +40.220, E3 +121188.328}
SPL {X  -162.820, Y  +632.362, Z    +0.000, E1   +62.930, E3 +121186.987}
SPL {X  -162.820, Y  +579.681, Z    +0.000, E1   +72.301, E3 +121202.774}
SPL {X  -162.820, Y  +408.049, Z    +0.000, E1   +72.202, E3 +121295.206}
ENDSPLINE

SPLINE
SPL {X  -162.820, Y  +452.249, Z    +0.000, E1   +66.666, E3 +121311.211}
ENDSPLINE

SPLINE
SPL {X  -162.820, Y  +427.408, Z    +0.000, E1   +67.534, E3 +121325.830}
SPL {X  -162.820, Y  +402.068, Z    +0.000, E1   +68.403, E3 +121339.891}
SPL {X  -162.804, Y  +378.229, Z    +0.000, E1   +69.183, E3 +121352.218}
SPL {X  -161.511, Y  +359.895, Z    +0.000, E1   +69.744, E3 +121361.510}
SPL {X  -158.246, Y  +342.178, Z    +0.000, E1   +70.136, E3 +121371.259}
SPL {X  -154.257, Y  +328.393, Z    +0.000, E1   +70.602, E3 +121377.052}
SPL {X  -150.447, Y  +318.243, Z    +0.000, E1   +70.683, E3 +121383.398}
SPL {X  -145.895, Y  +308.216, Z    +0.000, E1   +70.273, E3 +121393.351}
SPL {X  -140.654, Y  +298.483, Z    +0.000, E1   +69.615, E3 +121404.493}
SPL {X  -136.192, Y  +291.270, Z    +0.000, E1   +68.926, E3 +121413.457}
SPL {X  -131.963, Y  +285.127, Z    +0.000, E1   +68.405, E3 +121420.448}
SPL {X  -127.466, Y  +279.195, Z    +0.000, E1   +67.714, E3 +121427.735}
SPL {X  -119.204, Y  +269.591, Z    +0.000, E1   +69.726, E3 +121425.727}
SPL {X   -73.382, Y  +235.154, Z    +0.000, E1   +54.977, E3 +121591.404}
ENDSPLINE

SPLINE
SPL {X  -133.875, Y  +287.830, Z    +0.000, E1   +51.751, E3 +121730.606}
SPL {X  -153.240, Y  +325.474, Z    +0.000, E1   +39.999, E3 +121741.809}
SPL {X  -159.032, Y  +345.583, Z    +0.000, E1   +29.156, E3 +121742.293}
SPL {X  -161.304, Y  +358.334, Z    +0.000, E1   +20.524, E3 +121742.250}
SPL {X  -162.437, Y  +369.334, Z    +0.000, E1   +11.998, E3 +121743.429}
SPL {X  -162.814, Y  +379.161, Z    +0.000, E1    +3.343, E3 +121743.449}
SPL {X  -162.820, Y  +382.500, Z    +0.000, E1    +0.000, E3 +121742.931}
SPL {X  -162.820, Y  +384.390, Z    +0.000, E1    -3.279, E3 +121742.648}
SPL {X  -162.820, Y  +388.496, Z    +0.000, E1   -11.991, E3 +121742.550}
SPL {X  -162.820, Y  +392.944, Z    +0.000, E1   -22.020, E3 +121742.575}
SPL {X  -162.820, Y  +397.954, Z    +0.000, E1   -32.843, E3 +121742.615}
SPL {X  -162.820, Y  +404.232, Z    +0.000, E1   -44.157, E3 +121742.623}
SPL {X  -162.820, Y  +415.904, Z    +0.000, E1   -58.030, E3 +121742.897}
SPL {X  -162.820, Y  +467.484, Z    +0.000, E1   -73.355, E3 +121752.726}
SPL {X  -162.820, Y  +491.822, Z    +0.000, E1   -76.748, E3 +121754.149}
SPL {X  -162.820, Y  +654.572, Z    +0.000, E1   -72.288, E3 +121855.225}
SPL {X  -162.820, Y  +673.151, Z    +0.000, E1   -71.906, E3 +121871.794}
SPL {X  -161.514, Y  +694.081, Z    +0.000, E1   -71.845, E3 +121886.449}
SPL {X  -159.782, Y  +704.807, Z    +0.000, E1   -71.464, E3 +121897.431}
SPL {X  -157.050, Y  +716.463, Z    +0.000, E1   -71.316, E3 +121906.731}
SPL {X  -154.424, Y  +725.109, Z    +0.000, E1   -70.982, E3 +121915.583}
SPL {X  -150.493, Y  +735.646, Z    +0.000, E1   -70.534, E3 +121926.628}
SPL {X  -145.565, Y  +746.446, Z    +0.000, E1   -69.958, E3 +121938.337}
SPL {X  -141.153, Y  +754.655, Z    +0.000, E1   -69.344, E3 +121948.082}
SPL {X  -136.484, Y  +762.283, Z    +0.000, E1   -68.639, E3 +121957.714}
SPL {X  -132.373, Y  +768.304, Z    +0.000, E1   -68.109, E3 +121964.585}
SPL {X  -129.138, Y  +772.665, Z    +0.000, E1   -67.631, E3 +121969.932}
SPL {X  -125.533, Y  +777.190, Z    +0.000, E1   -67.475, E3 +121973.630}
SPL {X   -73.826, Y  +818.621, Z    +0.000, E1   -58.574, E3 +122069.122}
ENDSPLINE

SPLINE
SPL {X  -110.901, Y  +792.711, Z    +0.000, E1   -55.300, E3 +122253.980}
SPL {X  -144.508, Y  +748.519, Z    +0.000, E1   -46.961, E3 +122279.017}
SPL {X  -158.446, Y  +710.986, Z    +0.000, E1   -30.228, E3 +122282.382}
SPL {X  -162.035, Y  +689.470, Z    +0.000, E1   -15.657, E3 +122283.953}
SPL {X  -162.788, Y  +676.746, Z    +0.000, E1    -5.020, E3 +122283.860}
SPL {X  -162.820, Y  +671.525, Z    +0.000, E1    -0.042, E3 +122283.415}
SPL {X  -162.820, Y  +669.531, Z    +0.000, E1    +3.299, E3 +122283.103}
SPL {X  -162.820, Y  +664.807, Z    +0.000, E1   +13.064, E3 +122283.032}
SPL {X  -162.820, Y  +659.610, Z    +0.000, E1   +24.615, E3 +122283.013}
SPL {X  -162.820, Y  +651.281, Z    +0.000, E1   +40.220, E3 +122283.566}
SPL {X  -162.820, Y  +632.362, Z    +0.000, E1   +62.930, E3 +122282.225}
SPL {X  -162.820, Y  +579.681, Z    +0.000, E1   +72.301, E3 +122298.012}
SPL {X  -162.820, Y  +408.049, Z    +0.000, E1   +72.202, E3 +122390.444}
ENDSPLINE

SPLINE
SPL {X  -162.820, Y  +452.249, Z    +0.000, E1   +66.666, E3 +122406.449}
ENDSPLINE

SPLINE
SPL {X  -162.820, Y  +427.408, Z    +0.000, E1   +67.534, E3 +122421.068}
SPL {X  -162.820, Y  +402.068, Z    +0.000, E1   +68.403, E3 +122435.129}
SPL {X  -162.523, Y  +370.677, Z    +0.000, E1   +69.437, E3 +122451.190}
SPL {X  -158.958, Y  +345.247, Z    +0.000, E1   +70.087, E3 +122464.733}
SPL {X  -152.677, Y  +323.931, Z    +0.000, E1   +70.710, E3 +122474.494}
SPL {X  -148.063, Y  +312.768, Z    +0.000, E1   +70.492, E3 +122483.815}
SPL {X  -143.809, Y  +304.150, Z    +0.000, E1   +70.034, E3 +122492.958}
SPL {X  -139.938, Y  +297.268, Z    +0.000, E1   +69.438, E3 +122501.548}
SPL {X  -136.192, Y  +291.270, Z    +0.000, E1   +68.926, E3 +122508.695}
SPL {X  -131.963, Y  +285.127, Z    +0.000, E1   +68.405, E3 +122515.686}
SPL {X  -127.466, Y  +279.195, Z    +0.000, E1   +67.714, E3 +122522.973}
SPL {X  -119.204, Y  +269.591, Z    +0.000, E1   +69.726, E3 +122520.965}
SPL {X   -73.382, Y  +235.154, Z    +0.000, E1   +54.977, E3 +122686.642}
ENDSPLINE

SPLINE
SPL {X  -115.538, Y  +265.778, Z    +0.000, E1   +55.826, E3 +122817.093}
SPL {X  -140.740, Y  +298.630, Z    +0.000, E1   +48.901, E3 +122828.428}
SPL {X  -153.240, Y  +325.474, Z    +0.000, E1   +39.999, E3 +122837.047}
SPL {X  -160.567, Y  +353.506, Z    +0.000, E1   +24.043, E3 +122837.541}
SPL {X  -162.646, Y  +372.968, Z    +0.000, E1    +8.995, E3 +122838.718}
SPL {X  -162.820, Y  +382.382, Z    +0.000, E1    +0.204, E3 +122838.205}
SPL {X  -162.820, Y  +384.390, Z    +0.000, E1    -3.279, E3 +122837.886}
SPL {X  -162.820, Y  +388.496, Z    +0.000, E1   -11.991, E3 +122837.788}
SPL {X  -162.820, Y  +392.944, Z    +0.000, E1   -22.020, E3 +122837.813}
SPL {X  -162.820, Y  +397.954, Z    +0.000, E1   -32.843, E3 +122837.853}
SPL {X  -162.820, Y  +404.232, Z    +0.000, E1   -44.157, E3 +122837.861}
SPL {X  -162.820, Y  +415.904, Z    +0.000, E1   -58.030, E3 +122838.135}
SPL {X  -162.820, Y  +472.155, Z    +0.000, E1   -74.123, E3 +122848.238}
SPL {X  -162.820, Y  +661.743, Z    +0.000, E1   -73.395, E3 +122943.372}
ENDSPLINE

SPLINE
SPL {X  -162.820, Y  +658.105, Z    +0.000, E1   -71.889, E3 +122956.770}
ENDSPLINE

SPLINE
SPL {X  -162.784, Y  +676.927, Z    +0.000, E1   -71.815, E3 +122970.298}
SPL {X  -161.514, Y  +694.081, Z    +0.000, E1   -71.845, E3 +122981.687}
SPL {X  -159.782, Y  +704.807, Z    +0.000, E1   -71.464, E3 +122992.670}
SPL {X  -157.050, Y  +716.463, Z    +0.000, E1   -71.316, E3 +123001.969}
SPL {X  -154.424, Y  +725.109, Z    +0.000, E1   -70.982, E3 +123010.821}
SPL {X  -150.493, Y  +735.646, Z    +0.000, E1   -70.534, E3 +123021.866}
SPL {X  -145.565, Y  +746.446, Z    +0.000, E1   -69.958, E3 +123033.575}
SPL {X  -141.153, Y  +754.655, Z    +0.000, E1   -69.344, E3 +123043.320}
SPL {X  -136.484, Y  +762.283, Z    +0.000, E1   -68.639, E3 +123052.953}
SPL {X  -131.125, Y  +770.022, Z    +0.000, E1   -67.959, E3 +123061.859}
SPL {X  -126.438, Y  +776.086, Z    +0.000, E1   -67.465, E3 +123068.181}
SPL {X   -73.826, Y  +818.621, Z    +0.000, E1   -58.574, E3 +123164.361}
ENDSPLINE

SPLINE
SPL {X  -110.901, Y  +792.711, Z    +0.000, E1   -55.300, E3 +123349.218}
SPL {X  -144.508, Y  +748.519, Z    +0.000, E1   -46.961, E3 +123374.255}
SPL {X  -156.638, Y  +717.940, Z    +0.000, E1   -34.002, E3 +123376.991}
SPL {X  -160.830, Y  +698.875, Z    +0.000, E1   -22.517, E3 +123378.654}
SPL {X  -162.532, Y  +683.174, Z    +0.000, E1   -10.600, E3 +123379.260}
SPL {X  -162.820, Y  +671.472, Z    +0.000, E1    -0.171, E3 +123378.602}
SPL {X  -162.820, Y  +667.499, Z    +0.000, E1    +7.374, E3 +123378.343}
SPL {X  -162.820, Y  +663.777, Z    +0.000, E1   +15.496, E3 +123378.206}
SPL {X  -162.820, Y  +659.610, Z    +0.000, E1   +24.615, E3 +123378.251}
SPL {X  -162.820, Y  +651.281, Z    +0.000, E1   +40.220, E3 +123378.804}
SPL {X  -162.820, Y  +635.984, Z    +0.000, E1   +61.208, E3 +123376.458}
SPL {X  -162.820, Y  +617.261, Z    +0.000, E1   +67.803, E3 +123381.645}
SPL {X  -162.820, Y  +579.681, Z    +0.000, E1   +72.301, E3 +123393.250}
SPL {X  -162.820, Y  +408.049, Z    +0.000, E1   +72.202, E3 +123485.682}
ENDSPLINE

SPLINE
SPL {X  -162.820, Y  +452.249, Z    +0.000, E1   +66.666, E3 +123501.687}
ENDSPLINE

SPLINE
SPL {X  -162.820, Y  +427.408, Z    +0.000, E1   +67.534, E3 +123516.306}
SPL {X  -162.820, Y  +402.068, Z    +0.000, E1   +68.403, E3 +123530.367}
SPL {X  -162.804, Y  +378.229, Z    +0.000, E1   +69.183, E3 +123542.694}
SPL {X  -161.511, Y  +359.895, Z    +0.000, E1   +69.744, E3 +123551.986}
SPL {X  -158.246, Y  +342.178, Z    +0.000, E1   +70.136, E3 +123561.735}
SPL {X  -152.677, Y  +323.931, Z    +0.000, E1   +70.710, E3 +123569.732}
SPL {X  -148.063, Y  +312.768, Z    +0.000, E1   +70.492, E3 +123579.053}
SPL {X  -143.809, Y  +304.150, Z    +0.000, E1   +70.034, E3 +123588.196}
SPL {X  -139.938, Y  +297.268, Z    +0.000, E1   +69.438, E3 +123596.786}
SPL {X  -136.192, Y  +291.270, Z    +0.000, E1   +68.926, E3 +123603.934}
SPL {X  -132.794, Y  +286.287, Z    +0.000, E1   +68.653, E3 +123608.728}
SPL {X  -129.555, Y  +281.880, Z    +0.000, E1   +68.043, E3 +123614.828}
SPL {X  -126.523, Y  +278.020, Z    +0.000, E1   +67.371, E3 +123620.319}
SPL {X  -119.204, Y  +269.591, Z    +0.000, E1   +69.726, E3 +123616.203}
SPL {X   -73.382, Y  +235.154, Z    +0.000, E1   +54.977, E3 +123781.880}
ENDSPLINE

SPLINE
SPL {X  -133.875, Y  +287.830, Z    +0.000, E1   +51.751, E3 +123921.082}
SPL {X  -153.240, Y  +325.474, Z    +0.000, E1   +39.999, E3 +123932.285}
SPL {X  -159.032, Y  +345.583, Z    +0.000, E1   +29.156, E3 +123932.769}
SPL {X  -161.304, Y  +358.334, Z    +0.000, E1   +20.524, E3 +123932.727}
SPL {X  -162.437, Y  +369.334, Z    +0.000, E1   +11.998, E3 +123933.905}
SPL {X  -162.814, Y  +379.161, Z    +0.000, E1    +3.343, E3 +123933.925}
SPL {X  -162.820, Y  +382.751, Z    +0.000, E1    -0.252, E3 +123933.339}
SPL {X  -162.820, Y  +387.406, Z    +0.000, E1    -9.377, E3 +123933.060}
SPL {X  -162.820, Y  +392.944, Z    +0.000, E1   -22.020, E3 +123933.051}
SPL {X  -162.820, Y  +397.954, Z    +0.000, E1   -32.843, E3 +123933.091}
SPL {X  -162.820, Y  +404.232, Z    +0.000, E1   -44.157, E3 +123933.099}
SPL {X  -162.820, Y  +415.904, Z    +0.000, E1   -58.030, E3 +123933.373}
SPL {X  -162.820, Y  +472.155, Z    +0.000, E1   -74.123, E3 +123943.476}
SPL {X  -162.820, Y  +661.743, Z    +0.000, E1   -73.395, E3 +124038.610}
ENDSPLINE

SPLINE
SPL {X  -162.820, Y  +658.105, Z    +0.000, E1   -71.889, E3 +124052.008}
ENDSPLINE

SPLINE
SPL {X  -162.784, Y  +676.927, Z    +0.000, E1   -71.815, E3 +124065.536}
SPL {X  -161.514, Y  +694.081, Z    +0.000, E1   -71.845, E3 +124076.925}
SPL {X  -159.782, Y  +704.807, Z    +0.000, E1   -71.464, E3 +124087.908}
SPL {X  -157.050, Y  +716.463, Z    +0.000, E1   -71.316, E3 +124097.208}
SPL {X  -154.424, Y  +725.109, Z    +0.000, E1   -70.982, E3 +124106.059}
SPL {X  -151.195, Y  +733.918, Z    +0.000, E1   -70.611, E3 +124115.182}
SPL {X  -147.776, Y  +741.856, Z    +0.000, E1   -70.224, E3 +124123.630}
SPL {X  -144.623, Y  +748.297, Z    +0.000, E1   -69.772, E3 +124131.255}
SPL {X  -141.153, Y  +754.655, Z    +0.000, E1   -69.344, E3 +124138.558}
SPL {X  -136.484, Y  +762.283, Z    +0.000, E1   -68.639, E3 +124148.191}
SPL {X  -131.125, Y  +770.022, Z    +0.000, E1   -67.959, E3 +124157.097}
SPL {X  -126.438, Y  +776.086, Z    +0.000, E1   -67.465, E3 +124163.419}
SPL {X   -73.826, Y  +818.621, Z    +0.000, E1   -58.574, E3 +124259.599}
ENDSPLINE

SPLINE
SPL {X  -110.901, Y  +792.711, Z    +0.000, E1   -55.300, E3 +124444.457}
SPL {X  -144.508, Y  +748.519, Z    +0.000, E1   -46.961, E3 +124469.493}
SPL {X  -158.446, Y  +710.986, Z    +0.000, E1   -30.228, E3 +124472.858}
SPL {X  -162.035, Y  +689.470, Z    +0.000, E1   -15.657, E3 +124474.429}
SPL {X  -162.788, Y  +676.746, Z    +0.000, E1    -5.020, E3 +124474.337}
SPL {X  -162.820, Y  +671.525, Z    +0.000, E1    -0.042, E3 +124473.891}
SPL {X  -162.820, Y  +669.531, Z    +0.000, E1    +3.299, E3 +124473.580}
SPL {X  -162.820, Y  +664.807, Z    +0.000, E1   +13.064, E3 +124473.508}
SPL {X  -162.820, Y  +659.610, Z    +0.000, E1   +24.615, E3 +124473.489}
SPL {X  -162.820, Y  +651.281, Z    +0.000, E1   +40.220, E3 +124474.042}
SPL {X  -162.820, Y  +635.984, Z    +0.000, E1   +61.208, E3 +124471.696}
SPL {X  -162.820, Y  +617.261, Z    +0.000, E1   +67.803, E3 +124476.883}
SPL {X  -162.820, Y  +579.681, Z    +0.000, E1   +72.301, E3 +124488.488}
SPL {X  -162.820, Y  +408.049, Z    +0.000, E1   +72.202, E3 +124580.920}
ENDSPLINE

SPLINE
SPL {X  -162.820, Y  +452.249, Z    +0.000, E1   +66.666, E3 +124596.926}
ENDSPLINE

SPLINE
SPL {X  -162.820, Y  +427.408, Z    +0.000, E1   +67.534, E3 +124611.544}
SPL {X  -162.820, Y  +402.068, Z    +0.000, E1   +68.403, E3 +124625.605}
SPL {X  -162.523, Y  +370.677, Z    +0.000, E1   +69.437, E3 +124641.666}
SPL {X  -158.958, Y  +345.247, Z    +0.000, E1   +70.087, E3 +124655.209}
SPL {X  -154.257, Y  +328.393, Z    +0.000, E1   +70.602, E3 +124662.766}
SPL {X  -151.417, Y  +320.641, Z    +0.000, E1   +70.773, E3 +124666.649}
SPL {X  -148.063, Y  +312.768, Z    +0.000, E1   +70.492, E3 +124674.291}
SPL {X  -143.809, Y  +304.150, Z    +0.000, E1   +70.034, E3 +124683.434}
SPL {X  -139.938, Y  +297.268, Z    +0.000, E1   +69.438, E3 +124692.025}
SPL {X  -136.192, Y  +291.270, Z    +0.000, E1   +68.926, E3 +124699.172}
SPL {X  -131.963, Y  +285.127, Z    +0.000, E1   +68.405, E3 +124706.162}
SPL {X  -127.466, Y  +279.195, Z    +0.000, E1   +67.714, E3 +124713.450}
SPL {X  -119.204, Y  +269.591, Z    +0.000, E1   +69.726, E3 +124711.441}
SPL {X   -73.382, Y  +235.154, Z    +0.000, E1   +54.977, E3 +124877.118}
ENDSPLINE

SPLINE
SPL {X  -133.875, Y  +287.830, Z    +0.000, E1   +51.751, E3 +125016.320}
SPL {X  -153.240, Y  +325.474, Z    +0.000, E1   +39.999, E3 +125027.523}
SPL {X  -159.032, Y  +345.583, Z    +0.000, E1   +29.156, E3 +125028.008}
SPL {X  -161.304, Y  +358.334, Z    +0.000, E1   +20.524, E3 +125027.965}
SPL {X  -162.437, Y  +369.334, Z    +0.000, E1   +11.998, E3 +125029.143}
SPL {X  -162.814, Y  +379.161, Z    +0.000, E1    +3.343, E3 +125029.163}
SPL {X  -162.820, Y  +382.751, Z    +0.000, E1    -0.252, E3 +125028.577}
SPL {X  -162.820, Y  +387.406, Z    +0.000, E1    -9.377, E3 +125028.298}
SPL {X  -162.820, Y  +392.944, Z    +0.000, E1   -22.020, E3 +125028.289}
SPL {X  -162.820, Y  +397.954, Z    +0.000, E1   -32.843, E3 +125028.329}
SPL {X  -162.820, Y  +404.232, Z    +0.000, E1   -44.157, E3 +125028.337}
SPL {X  -162.820, Y  +415.904, Z    +0.000, E1   -58.030, E3 +125028.611}
SPL {X  -162.820, Y  +467.484, Z    +0.000, E1   -73.355, E3 +125038.440}
SPL {X  -162.820, Y  +491.822, Z    +0.000, E1   -76.748, E3 +125039.864}
SPL {X  -162.820, Y  +661.743, Z    +0.000, E1   -73.395, E3 +125133.848}
ENDSPLINE

SPLINE
SPL {X  -162.820, Y  +658.105, Z    +0.000, E1   -71.889, E3 +125147.246}
ENDSPLINE

SPLINE
SPL {X  -162.784, Y  +676.927, Z    +0.000, E1   -71.815, E3 +125160.774}
SPL {X  -161.514, Y  +694.081, Z    +0.000, E1   -71.845, E3 +125172.163}
SPL {X  -159.782, Y  +704.807, Z    +0.000, E1   -71.464, E3 +125183.146}
SPL {X  -157.050, Y  +716.463, Z    +0.000, E1   -71.316, E3 +125192.446}
SPL {X  -154.424, Y  +725.109, Z    +0.000, E1   -70.982, E3 +125201.298}
SPL {X  -151.195, Y  +733.918, Z    +0.000, E1   -70.611, E3 +125210.420}
SPL {X  -147.776, Y  +741.856, Z    +0.000, E1   -70.224, E3 +125218.868}
SPL {X  -143.411, Y  +750.594, Z    +0.000, E1   -69.653, E3 +125229.024}
SPL {X  -138.205, Y  +759.580, Z    +0.000, E1   -68.913, E3 +125239.973}
SPL {X  -133.334, Y  +766.947, Z    +0.000, E1   -68.226, E3 +125248.839}
SPL {X  -129.138, Y  +772.665, Z    +0.000, E1   -67.631, E3 +125255.646}
SPL {X  -125.533, Y  +777.190, Z    +0.000, E1   -67.475, E3 +125259.344}
SPL {X   -73.826, Y  +818.621, Z    +0.000, E1   -58.574, E3 +125354.837}
ENDSPLINE

SPLINE
SPL {X  -110.901, Y  +792.711, Z    +0.000, E1   -55.300, E3 +125539.695}
SPL {X  -144.508, Y  +748.519, Z    +0.000, E1   -46.961, E3 +125564.731}
SPL {X  -156.638, Y  +717.940, Z    +0.000, E1   -34.002, E3 +125567.467}
SPL {X  -160.830, Y  +698.875, Z    +0.000, E1   -22.517, E3 +125569.131}
SPL {X  -162.532, Y  +683.174, Z    +0.000, E1   -10.600, E3 +125569.736}
SPL {X  -162.820, Y  +671.754, Z    +0.000, E1    -0.424, E3 +125569.152}
SPL {X  -162.820, Y  +669.531, Z    +0.000, E1    +3.299, E3 +125568.818}
SPL {X  -162.820, Y  +664.807, Z    +0.000, E1   +13.064, E3 +125568.746}
SPL {X  -162.820, Y  +659.610, Z    +0.000, E1   +24.615, E3 +125568.727}
SPL {X  -162.820, Y  +651.281, Z    +0.000, E1   +40.220, E3 +125569.280}
SPL {X  -162.820, Y  +632.362, Z    +0.000, E1   +62.930, E3 +125567.940}
SPL {X  -162.820, Y  +579.681, Z    +0.000, E1   +72.301, E3 +125583.726}
SPL {X  -162.820, Y  +408.049, Z    +0.000, E1   +72.202, E3 +125676.158}
ENDSPLINE

SPLINE
SPL {X  -162.820, Y  +452.249, Z    +0.000, E1   +66.666, E3 +125692.164}
ENDSPLINE

SPLINE
SPL {X  -162.820, Y  +427.408, Z    +0.000, E1   +67.534, E3 +125706.782}
SPL {X  -162.820, Y  +402.068, Z    +0.000, E1   +68.403, E3 +125720.844}
SPL {X  -162.523, Y  +370.677, Z    +0.000, E1   +69.437, E3 +125736.904}
SPL {X  -158.958, Y  +345.247, Z    +0.000, E1   +70.087, E3 +125750.447}
SPL {X  -152.677, Y  +323.931, Z    +0.000, E1   +70.710, E3 +125760.208}
SPL {X  -148.063, Y  +312.768, Z    +0.000, E1   +70.492, E3 +125769.529}
SPL {X  -143.809, Y  +304.150, Z    +0.000, E1   +70.034, E3 +125778.672}
SPL {X  -139.938, Y  +297.268, Z    +0.000, E1   +69.438, E3 +125787.263}
SPL {X  -136.192, Y  +291.270, Z    +0.000, E1   +68.926, E3 +125794.410}
SPL {X  -132.794, Y  +286.287, Z    +0.000, E1   +68.653, E3 +125799.205}
SPL {X  -129.555, Y  +281.880, Z    +0.000, E1   +68.043, E3 +125805.304}
SPL {X  -126.523, Y  +278.020, Z    +0.000, E1   +67.371, E3 +125810.796}
SPL {X  -119.204, Y  +269.591, Z    +0.000, E1   +69.726, E3 +125806.679}
SPL {X   -73.382, Y  +235.154, Z    +0.000, E1   +54.977, E3 +125972.356}
ENDSPLINE

SPLINE
SPL {X  -133.875, Y  +287.830, Z    +0.000, E1   +51.751, E3 +126111.558}
SPL {X  -153.240, Y  +325.474, Z    +0.000, E1   +39.999, E3 +126122.761}
SPL {X  -159.032, Y  +345.583, Z    +0.000, E1   +29.156, E3 +126123.246}
SPL {X  -161.304, Y  +358.334, Z    +0.000, E1   +20.524, E3 +126123.203}
SPL {X  -162.437, Y  +369.334, Z    +0.000, E1   +11.998, E3 +126124.382}
SPL {X  -162.814, Y  +379.161, Z    +0.000, E1    +3.343, E3 +126124.401}
SPL {X  -162.820, Y  +382.500, Z    +0.000, E1    +0.000, E3 +126123.883}
SPL {X  -162.820, Y  +384.390, Z    +0.000, E1    -3.279, E3 +126123.601}
SPL {X  -162.820, Y  +388.496, Z    +0.000, E1   -11.991, E3 +126123.502}
SPL {X  -162.820, Y  +392.944, Z    +0.000, E1   -22.020, E3 +126123.527}
SPL {X  -162.820, Y  +397.954, Z    +0.000, E1   -32.843, E3 +126123.567}
SPL {X  -162.820, Y  +404.232, Z    +0.000, E1   -44.157, E3 +126123.575}
SPL {X  -162.820, Y  +415.904, Z    +0.000, E1   -58.030, E3 +126123.849}
SPL {X  -162.820, Y  +472.155, Z    +0.000, E1   -74.123, E3 +126133.952}
SPL {X  -162.820, Y  +654.572, Z    +0.000, E1   -72.288, E3 +126236.177}
SPL {X  -162.820, Y  +673.151, Z    +0.000, E1   -71.906, E3 +126252.747}
SPL {X  -161.514, Y  +694.081, Z    +0.000, E1   -71.845, E3 +126267.402}
SPL {X  -159.782, Y  +704.807, Z    +0.000, E1   -71.464, E3 +126278.384}
SPL {X  -157.050, Y  +716.463, Z    +0.000, E1   -71.316, E3 +126287.684}
SPL {X  -154.424, Y  +725.109, Z    +0.000, E1   -70.982, E3 +126296.536}
SPL {X  -150.493, Y  +735.646, Z    +0.000, E1   -70.534, E3 +126307.580}
SPL {X  -145.565, Y  +746.446, Z    +0.000, E1   -69.958, E3 +126319.289}
SPL {X  -142.097, Y  +752.991, Z    +0.000, E1   -69.463, E3 +126327.029}
SPL {X  -138.205, Y  +759.580, Z    +0.000, E1   -68.913, E3 +126335.211}
SPL {X  -133.334, Y  +766.947, Z    +0.000, E1   -68.226, E3 +126344.077}
SPL {X  -129.138, Y  +772.665, Z    +0.000, E1   -67.631, E3 +126350.884}
SPL {X  -125.533, Y  +777.190, Z    +0.000, E1   -67.475, E3 +126354.582}
SPL {X   -75.773, Y  +817.614, Z    +0.000, E1   -59.878, E3 +126435.547}
SPL {X   -71.637, Y  +819.714, Z    +0.000, E1   -56.371, E3 +126481.154}
ENDSPLINE

SPLINE
SPL {X  -110.901, Y  +792.711, Z    +0.000, E1   -55.300, E3 +126634.933}
SPL {X  -144.508, Y  +748.519, Z    +0.000, E1   -46.961, E3 +126659.969}
SPL {X  -158.446, Y  +710.986, Z    +0.000, E1   -30.228, E3 +126663.334}
SPL {X  -162.035, Y  +689.470, Z    +0.000, E1   -15.657, E3 +126664.905}
SPL {X  -162.788, Y  +676.746, Z    +0.000, E1    -5.020, E3 +126664.813}
SPL {X  -162.820, Y  +671.525, Z    +0.000, E1    -0.042, E3 +126664.367}
SPL {X  -162.820, Y  +669.531, Z    +0.000, E1    +3.299, E3 +126664.056}
SPL {X  -162.820, Y  +664.807, Z    +0.000, E1   +13.064, E3 +126663.984}
SPL {X  -162.820, Y  +659.610, Z    +0.000, E1   +24.615, E3 +126663.965}
SPL {X  -162.820, Y  +651.281, Z    +0.000, E1   +40.220, E3 +126664.518}
SPL {X  -162.820, Y  +632.362, Z    +0.000, E1   +62.930, E3 +126663.178}
SPL {X  -162.820, Y  +579.681, Z    +0.000, E1   +72.301, E3 +126678.964}
SPL {X  -162.820, Y  +408.049, Z    +0.000, E1   +72.202, E3 +126771.396}
ENDSPLINE

SPLINE
SPL {X  -162.820, Y  +452.249, Z    +0.000, E1   +66.666, E3 +126787.402}
ENDSPLINE

SPLINE
SPL {X  -162.820, Y  +427.408, Z    +0.000, E1   +67.534, E3 +126802.020}
SPL {X  -162.820, Y  +402.068, Z    +0.000, E1   +68.403, E3 +126816.082}
SPL {X  -162.523, Y  +370.677, Z    +0.000, E1   +69.437, E3 +126832.142}
SPL {X  -158.958, Y  +345.247, Z    +0.000, E1   +70.087, E3 +126845.685}
SPL {X  -152.677, Y  +323.931, Z    +0.000, E1   +70.710, E3 +126855.446}
SPL {X  -148.063, Y  +312.768, Z    +0.000, E1   +70.492, E3 +126864.768}
SPL {X  -143.809, Y  +304.150, Z    +0.000, E1   +70.034, E3 +126873.910}
SPL {X  -139.938, Y  +297.268, Z    +0.000, E1   +69.438, E3 +126882.501}
SPL {X  -136.192, Y  +291.270, Z    +0.000, E1   +68.926, E3 +126889.648}
SPL {X  -132.794, Y  +286.287, Z    +0.000, E1   +68.653, E3 +126894.443}
SPL {X  -129.555, Y  +281.880, Z    +0.000, E1   +68.043, E3 +126900.543}
SPL {X  -126.523, Y  +278.020, Z    +0.000, E1   +67.371, E3 +126906.034}
SPL {X  -119.204, Y  +269.591, Z    +0.000, E1   +69.726, E3 +126901.917}
SPL {X   -73.382, Y  +235.154, Z    +0.000, E1   +54.977, E3 +127067.594}
ENDSPLINE

SPLINE
SPL {X  -133.875, Y  +287.830, Z    +0.000, E1   +51.751, E3 +127206.796}
SPL {X  -153.240, Y  +325.474, Z    +0.000, E1   +39.999, E3 +127218.000}
SPL {X  -160.567, Y  +353.506, Z    +0.000, E1   +24.043, E3 +127218.494}
SPL {X  -162.646, Y  +372.968, Z    +0.000, E1    +8.995, E3 +127219.670}
SPL {X  -162.820, Y  +382.382, Z    +0.000, E1    +0.204, E3 +127219.157}
SPL {X  -162.820, Y  +384.390, Z    +0.000, E1    -3.279, E3 +127218.839}
SPL {X  -162.820, Y  +388.496, Z    +0.000, E1   -11.991, E3 +127218.740}
SPL {X  -162.820, Y  +392.944, Z    +0.000, E1   -22.020, E3 +127218.765}
SPL {X  -162.820, Y  +397.954, Z    +0.000, E1   -32.843, E3 +127218.805}
SPL {X  -162.820, Y  +404.232, Z    +0.000, E1   -44.157, E3 +127218.814}
SPL {X  -162.820, Y  +415.904, Z    +0.000, E1   -58.030, E3 +127219.087}
SPL {X  -162.820, Y  +472.155, Z    +0.000, E1   -74.123, E3 +127229.190}
SPL {X  -162.820, Y  +661.743, Z    +0.000, E1   -73.395, E3 +127324.324}
ENDSPLINE

SPLINE
SPL {X  -162.820, Y  +658.105, Z    +0.000, E1   -71.889, E3 +127337.722}
ENDSPLINE

SPLINE
SPL {X  -162.784, Y  +676.927, Z    +0.000, E1   -71.815, E3 +127351.250}
SPL {X  -161.514, Y  +694.081, Z    +0.000, E1   -71.845, E3 +127362.640}
SPL {X  -159.782, Y  +704.807, Z    +0.000, E1   -71.464, E3 +127373.622}
SPL {X  -157.050, Y  +716.463, Z    +0.000, E1   -71.316, E3 +127382.922}
SPL {X  -154.424, Y  +725.109, Z    +0.000, E1   -70.982, E3 +127391.774}
SPL {X  -150.493, Y  +735.646, Z    +0.000, E1   -70.534, E3 +127402.819}
SPL {X  -145.565, Y  +746.446, Z    +0.000, E1   -69.958, E3 +127414.527}
SPL {X  -141.153, Y  +754.655, Z    +0.000, E1   -69.344, E3 +127424.272}
SPL {X  -137.365, Y  +760.914, Z    +0.000, E1   -68.751, E3 +127432.211}
SPL {X  -133.334, Y  +766.947, Z    +0.000, E1   -68.226, E3 +127439.315}
SPL {X  -129.138, Y  +772.665, Z    +0.000, E1   -67.631, E3 +127446.122}
SPL {X  -125.533, Y  +777.190, Z    +0.000, E1   -67.475, E3 +127449.820}
SPL {X   -73.826, Y  +818.621, Z    +0.000, E1   -58.574, E3 +127545.313}
ENDSPLINE

SPLINE
SPL {X  -110.901, Y  +792.711, Z    +0.000, E1   -55.300, E3 +127730.171}
SPL {X  -144.508, Y  +748.519, Z    +0.000, E1   -46.961, E3 +127755.207}
SPL {X  -158.446, Y  +710.986, Z    +0.000, E1   -30.228, E3 +127758.572}
SPL {X  -162.035, Y  +689.470, Z    +0.000, E1   -15.657, E3 +127760.143}
SPL {X  -162.788, Y  +676.746, Z    +0.000, E1    -5.020, E3 +127760.051}
SPL {X  -162.820, Y  +671.525, Z    +0.000, E1    -0.042, E3 +127759.605}
SPL {X  -162.820, Y  +670.529, Z    +0.000, E1    +1.628, E3 +127759.307}
SPL {X  -162.820, Y  +667.499, Z    +0.000, E1    +7.374, E3 +127759.295}
SPL {X  -162.820, Y  +663.777, Z    +0.000, E1   +15.496, E3 +127759.158}
SPL {X  -162.820, Y  +659.610, Z    +0.000, E1   +24.615, E3 +127759.204}
SPL {X  -162.820, Y  +651.281, Z    +0.000, E1   +40.220, E3 +127759.757}
SPL {X  -162.820, Y  +632.362, Z    +0.000, E1   +62.930, E3 +127758.416}
SPL {X  -162.820, Y  +579.681, Z    +0.000, E1   +72.301, E3 +127774.202}
SPL {X  -162.820, Y  +408.049, Z    +0.000, E1   +72.202, E3 +127866.634}
ENDSPLINE

SPLINE
SPL {X  -162.820, Y  +459.124, Z    +0.000, E1   +66.408, E3 +127878.406}
ENDSPLINE

SPLINE
SPL {X  -162.820, Y  +444.776, Z    +0.000, E1   +66.898, E3 +127887.298}
SPL {X  -162.820, Y  +427.408, Z    +0.000, E1   +67.534, E3 +127897.258}
SPL {X  -162.820, Y  +409.075, Z    +0.000, E1   +68.145, E3 +127907.643}
SPL {X  -162.820, Y  +384.968, Z    +0.000, E1   +68.973, E3 +127920.202}
SPL {X  -162.073, Y  +364.922, Z    +0.000, E1   +69.599, E3 +127930.327}
SPL {X  -158.958, Y  +345.247, Z    +0.000, E1   +70.087, E3 +127940.923}
SPL {X  -154.257, Y  +328.393, Z    +0.000, E1   +70.602, E3 +127948.480}
SPL {X  -150.447, Y  +318.243, Z    +0.000, E1   +70.683, E3 +127954.827}
SPL {X  -147.136, Y  +310.777, Z    +0.000, E1   +70.431, E3 +127961.726}
SPL {X  -143.809, Y  +304.150, Z    +0.000, E1   +70.034, E3 +127969.148}
SPL {X  -139.938, Y  +297.268, Z    +0.000, E1   +69.438, E3 +127977.739}
SPL {X  -136.192, Y  +291.270, Z    +0.000, E1   +68.926, E3 +127984.886}
SPL {X  -131.963, Y  +285.127, Z    +0.000, E1   +68.405, E3 +127991.876}
SPL {X  -127.466, Y  +279.195, Z    +0.000, E1   +67.714, E3 +127999.164}
SPL {X  -119.204, Y  +269.591, Z    +0.000, E1   +69.726, E3 +127997.155}
SPL {X   -73.382, Y  +235.154, Z    +0.000, E1   +54.977, E3 +128162.832}
ENDSPLINE

SPLINE
SPL {X  -115.538, Y  +265.778, Z    +0.000, E1   +55.826, E3 +128293.283}
SPL {X  -140.740, Y  +298.630, Z    +0.000, E1   +48.901, E3 +128304.619}
SPL {X  -153.240, Y  +325.474, Z    +0.000, E1   +39.999, E3 +128313.238}
SPL {X  -160.567, Y  +353.506, Z    +0.000, E1   +24.043, E3 +128313.732}
SPL {X  -162.646, Y  +372.968, Z    +0.000, E1    +8.995, E3 +128314.909}
SPL {X  -162.820, Y  +382.646, Z    +0.000, E1    -0.044, E3 +128314.323}
SPL {X  -162.820, Y  +387.406, Z    +0.000, E1    -9.377, E3 +128314.012}
SPL {X  -162.820, Y  +392.944, Z    +0.000, E1   -22.020, E3 +128314.003}
SPL {X  -162.820, Y  +397.954, Z    +0.000, E1   -32.843, E3 +128314.044}
SPL {X  -162.820, Y  +404.232, Z    +0.000, E1   -44.157, E3 +128314.052}
SPL {X  -162.820, Y  +415.904, Z    +0.000, E1   -58.030, E3 +128314.325}
SPL {X  -162.820, Y  +472.155, Z    +0.000, E1   -74.123, E3 +128324.428}
SPL {X  -162.820, Y  +661.743, Z    +0.000, E1   -73.395, E3 +128419.562}
ENDSPLINE

SPLINE
SPL {X  -162.820, Y  +658.105, Z    +0.000, E1   -71.889, E3 +128432.960}
ENDSPLINE

SPLINE
SPL {X  -162.784, Y  +676.927, Z    +0.000, E1   -71.815, E3 +128446.488}
SPL {X  -161.514, Y  +694.081, Z    +0.000, E1   -71.845, E3 +128457.878}
SPL {X  -159.782, Y  +704.807, Z    +0.000, E1   -71.464, E3 +128468.860}
SPL {X  -157.050, Y  +716.463, Z    +0.000, E1   -71.316, E3 +128478.160}
SPL {X  -154.424, Y  +725.109, Z    +0.000, E1   -70.982, E3 +128487.012}
SPL {X  -151.195, Y  +733.918, Z    +0.000, E1   -70.611, E3 +128496.134}
SPL {X  -147.776, Y  +741.856, Z    +0.000, E1   -70.224, E3 +128504.582}
SPL {X  -144.623, Y  +748.297, Z    +0.000, E1   -69.772, E3 +128512.207}
SPL {X  -141.153, Y  +754.655, Z    +0.000, E1   -69.344, E3 +128519.511}
SPL {X  -137.365, Y  +760.914, Z    +0.000, E1   -68.751, E3 +128527.449}
SPL {X  -133.334, Y  +766.947, Z    +0.000, E1   -68.226, E3 +128534.554}
SPL {X  -129.138, Y  +772.665, Z    +0.000, E1   -67.631, E3 +128541.360}
SPL {X  -125.533, Y  +777.190, Z    +0.000, E1   -67.475, E3 +128545.058}
SPL {X   -73.826, Y  +818.621, Z    +0.000, E1   -58.574, E3 +128640.551}
ENDSPLINE

SPLINE
SPL {X  -110.901, Y  +792.711, Z    +0.000, E1   -55.300, E3 +128825.409}
SPL {X  -144.508, Y  +748.519, Z    +0.000, E1   -46.961, E3 +128850.445}
SPL {X  -158.446, Y  +710.986, Z    +0.000, E1   -30.228, E3 +128853.811}
SPL {X  -162.035, Y  +689.470, Z    +0.000, E1   -15.657, E3 +128855.381}
SPL {X  -162.788, Y  +676.746, Z    +0.000, E1    -5.020, E3 +128855.289}
SPL {X  -162.820, Y  +671.525, Z    +0.000, E1    -0.042, E3 +128854.843}
SPL {X  -162.820, Y  +669.531, Z    +0.000, E1    +3.299, E3 +128854.532}
SPL {X  -162.820, Y  +664.807, Z    +0.000, E1   +13.064, E3 +128854.461}
SPL {X  -162.820, Y  +659.610, Z    +0.000, E1   +24.615, E3 +128854.442}
SPL {X  -162.820, Y  +651.281, Z    +0.000, E1   +40.220, E3 +128854.995}
SPL {X  -162.820, Y  +635.984, Z    +0.000, E1   +61.208, E3 +128852.649}
SPL {X  -162.820, Y  +617.261, Z    +0.000, E1   +67.803, E3 +128857.835}
SPL {X  -162.820, Y  +579.681, Z    +0.000, E1   +72.301, E3 +128869.440}
SPL {X  -162.820, Y  +408.049, Z    +0.000, E1   +72.202, E3 +128961.872}
ENDSPLINE

SPLINE
SPL {X  -162.820, Y  +452.249, Z    +0.000, E1   +66.666, E3 +128977.878}
ENDSPLINE

SPLINE
SPL {X  -162.820, Y  +427.408, Z    +0.000, E1   +67.534, E3 +128992.496}
SPL {X  -162.820, Y  +409.075, Z    +0.000, E1   +68.145, E3 +129002.881}
SPL {X  -162.820, Y  +384.968, Z    +0.000, E1   +68.973, E3 +129015.440}
SPL {X  -161.511, Y  +359.895, Z    +0.000, E1   +69.744, E3 +129028.177}
SPL {X  -158.246, Y  +342.178, Z    +0.000, E1   +70.136, E3 +129037.926}
SPL {X  -152.677, Y  +323.931, Z    +0.000, E1   +70.710, E3 +129045.923}
ENDSPLINE

SPLINE
SPL {X  -153.052, Y  +324.954, Z    +0.000, E1   +68.671, E3 +129061.572}
ENDSPLINE

SPLINE
SPL {X  -149.405, Y  +315.782, Z    +0.000, E1   +68.161, E3 +129072.337}
SPL {X  -145.408, Y  +307.240, Z    +0.000, E1   +67.667, E3 +129082.316}
SPL {X  -141.308, Y  +299.614, Z    +0.000, E1   +67.079, E3 +129091.842}
SPL {X  -137.907, Y  +293.943, Z    +0.000, E1   +66.608, E3 +129098.821}
SPL {X  -134.802, Y  +289.183, Z    +0.000, E1   +66.143, E3 +129104.957}
SPL {X  -131.727, Y  +284.801, Z    +0.000, E1   +65.590, E3 +129110.971}
SPL {X  -128.890, Y  +281.012, Z    +0.000, E1   +65.392, E3 +129114.717}
SPL {X  -121.325, Y  +271.915, Z    +0.000, E1   +67.092, E3 +129114.283}
SPL {X   -79.997, Y  +238.687, Z    +0.000, E1   +54.340, E3 +129273.039}
ENDSPLINE

SPLINE
SPL {X  -139.099, Y  +295.872, Z    +0.000, E1   +47.860, E3 +129400.915}
SPL {X  -156.463, Y  +335.448, Z    +0.000, E1   +33.333, E3 +129411.623}
SPL {X  -161.312, Y  +358.394, Z    +0.000, E1   +19.478, E3 +129413.257}
SPL {X  -162.549, Y  +371.111, Z    +0.000, E1    +9.905, E3 +129413.317}
SPL {X  -162.818, Y  +379.769, Z    +0.000, E1    +2.607, E3 +129413.059}
SPL {X  -162.820, Y  +382.500, Z    +0.000, E1    +0.000, E3 +129412.629}
SPL {X  -162.820, Y  +383.721, Z    +0.000, E1    -1.897, E3 +129412.366}
SPL {X  -162.820, Y  +387.689, Z    +0.000, E1    -9.147, E3 +129412.263}
SPL {X  -162.820, Y  +392.805, Z    +0.000, E1   -19.930, E3 +129412.236}
SPL {X  -162.820, Y  +397.742, Z    +0.000, E1   -30.068, E3 +129412.268}
SPL {X  -162.820, Y  +403.938, Z    +0.000, E1   -41.112, E3 +129412.248}
SPL {X  -162.820, Y  +415.430, Z    +0.000, E1   -55.307, E3 +129412.447}
SPL {X  -162.820, Y  +466.986, Z    +0.000, E1   -71.397, E3 +129424.206}
SPL {X  -162.820, Y  +661.594, Z    +0.000, E1   -73.988, E3 +129509.832}
ENDSPLINE

SPLINE
SPL {X  -162.820, Y  +646.360, Z    +0.000, E1   -70.938, E3 +129530.963}
ENDSPLINE

SPLINE
SPL {X  -162.820, Y  +667.477, Z    +0.000, E1   -70.889, E3 +129546.478}
SPL {X  -162.462, Y  +684.286, Z    +0.000, E1   -70.880, E3 +129558.711}
SPL {X  -160.799, Y  +699.074, Z    +0.000, E1   -70.750, E3 +129570.575}
SPL {X  -158.733, Y  +709.754, Z    +0.000, E1   -70.504, E3 +129580.458}
SPL {X  -156.566, Y  +718.194, Z    +0.000, E1   -70.115, E3 +129589.939}
SPL {X  -153.268, Y  +728.449, Z    +0.000, E1   -69.855, E3 +129599.565}
SPL {X  -150.033, Y  +736.750, Z    +0.000, E1   -69.498, E3 +129608.276}
SPL {X  -146.704, Y  +744.128, Z    +0.000, E1   -68.985, E3 +129617.398}
SPL {X  -143.061, Y  +751.243, Z    +0.000, E1   -68.459, E3 +129626.094}
SPL {X  -139.143, Y  +758.055, Z    +0.000, E1   -68.038, E3 +129633.657}
SPL {X  -134.977, Y  +764.558, Z    +0.000, E1   -67.353, E3 +129642.228}
SPL {X  -130.728, Y  +770.560, Z    +0.000, E1   -66.612, E3 +129650.263}
SPL {X  -125.283, Y  +777.493, Z    +0.000, E1   -66.879, E3 +129653.988}
SPL {X   -78.323, Y  +816.244, Z    +0.000, E1   -56.979, E3 +129761.084}
ENDSPLINE

